(* Logix 5000 project; controller E2122_083_261121_V1 vendor 1 type 14 code 196 rev 32.11; software revision 32.00 *)

TASK MainTask (continuous, watchdog 500 ms) : MainProgram

MODULES
   Local : vendor 1 type 14 code 196 (5069 0, rev 32.11)
      HP : vendor 1 type 14 code 149 (Ethernet 192.168.4.220, rev 24.1, $01a7d3c3$ RPI 20 ms, $5cc36044$ RPI 20 ms, $f3259996$ RPI 20 ms, $494006c6$ RPI 20 ms, $5c112d50$ RPI 20 ms, $6e423aaa$ RPI 20 ms, $f0f89954$ RPI 20 ms, $571546d8$ RPI 20 ms, $782664ef$ RPI 20 ms, $0e272f01$ RPI 20 ms, $e1a11e23$ RPI 20 ms)
      RFID : vendor 322 type 12 code 102 (Ethernet 192.168.4.79, rev 1.1, StandardDataDriven RPI 10 ms)
      RFID_2 : vendor 322 type 12 code 102 (Ethernet 192.168.4.80, rev 1.1, StandardDataDriven RPI 10 ms)
       : 5069-IB16 (5069 1, rev 2.1, StandardDataDriven RPI 5 ms)
       : 5069-OB16 (5069 2, rev 2.1, StandardDataDriven RPI 5 ms)
END_MODULES

TYPE Createparams :
STRUCT
   Type : DINT;   // 1 for TCP , 2 for UDP
   Addr : SockAddr;
END_STRUCT
END_TYPE

TYPE OpenconnParams :
STRUCT
   Timeout : DINT;
   DestAddr : STRING;
END_STRUCT
END_TYPE

TYPE SOCK_Addr :
STRUCT
   Family : INT;   // Address Family Must be 2
   Port : INT;   // Port Number
   Addr : SINT[4];   // IP Address
END_STRUCT
END_TYPE

TYPE SOCK_CreateParams :
STRUCT
   Type : DINT;   // 1 - TCP 2- UPD
   Addr : SOCK_Addr;
END_STRUCT
END_TYPE

TYPE SOCK_DATA_CLIENT :
STRUCT
   Create_Source : SOCK_CreateParams;
   Instance : DINT;
   Connect_Source : SOCK_OpenConnParam;
   Read_Source : SOCK_ReadParams;
   Read_Response : SOCK_ReadResponse;
   Write_Source : SOCK_WriteParams;
   Write_SizeSent : DINT;
END_STRUCT
END_TYPE

TYPE SOCK_OpenConnParam :
STRUCT
   Timeout : DINT;
   DestAddr : STRING;
END_STRUCT
END_TYPE

TYPE SOCK_ReadParams :
STRUCT
   Timeout : DINT;
   BufLen : DINT;
END_STRUCT
END_TYPE

TYPE SOCK_ReadResponse :
STRUCT
   FromAddr : SOCK_Addr;
   Buffer : STRING_READBUFFER;
END_STRUCT
END_TYPE

TYPE SOCK_WriteParams :
STRUCT
   Timeout : DINT;
   ToAddr : SOCK_Addr;
   Buffer : STRING_WRITEBUFFER;
END_STRUCT
END_TYPE

TYPE SockAddr :
STRUCT
   Family : INT;   // 2 for IP4 family
   Port : INT;   // Port number
   Addr : DINT;   // Local IP = 0
END_STRUCT
END_TYPE

TYPE STR_480 :
STRUCT
   LEN : DINT;
   DATA : SINT[82];
END_STRUCT
END_TYPE

TYPE STRING_READBUFFER :
STRUCT
   LEN : DINT;
   DATA : SINT[484];
END_STRUCT
END_TYPE

TYPE STRING_WRITEBUFFER :
STRUCT
   LEN : DINT;
   DATA : SINT[462];
END_STRUCT
END_TYPE

TYPE WriteParams :
STRUCT
   Timeout : DINT;
   ToAddr : SockAddr;
   Buf : STR_480;
END_STRUCT
END_TYPE

ADD_ON_INSTRUCTION INACTIVE   (* revision 2.4 *)
VAR_INPUT
   iiChannelNo : INT; {required}   // channel-No. of DTE102
   ixConnOK : BOOL; {required}   // Ethernet/IP connection to DTE102 is OK
END_VAR
VAR_IN_OUT
   iarbDTE102 : SINT[80]; {required}   // input data from DTE102
   oarbDTE102 : SINT[80]; {required}   // output data to DTE102
END_VAR
VAR_INPUT
   ixAckDiag : BOOL; {required}   // acknowledge diagnostic data
END_VAR
VAR_OUTPUT
   oiDiagLength : INT; {access Read Only, required}   // number of diagnostic data
END_VAR
VAR_IN_OUT
   oardwDiagData : DINT[4]; {required}   // diagnostic data
END_VAR
VAR
   IChannelNo : INT; {access None}   // channel-No. set by ConnOK
   IActInputSize : INT; {access None}   // actual input data size of DTE102
   XConnOK : BOOL; {access None}   // connection OK
   IActOutputSize : INT; {access None}   // actual output data size of DTE102
   IDataOffset : INT; {access None}   // offset in DTE data
   XreIxAckDiag : BOOL; {access None}   // rising edge input acknowledge diagnostic data
   XprevIxAckDiag : BOOL; {access None}   // previous state of input acknowledge diagnostic data
   XInitDiag : BOOL; {access None}   // initialize output diagnostic data
   bStatusDTE : SINT; {access None}
   IRdIdx : INT; {access None}   // read index pointer
   XDrRdy : BOOL; {access None}   // read diagnostic data finished
   XDiag : BOOL; {access None}   // unread diagnostic data available
   IWrIdx : INT; {access None}   // write index pointer
END_VAR

ROUTINE Logic   (* structured text *)
   (*Disclaimer of Warranties
   ifm disclaims to the fullest extent authorized by law any and all warranties, whether express or implied, including,
   without limitation, any implied warranties of title, non-infringement, quiet enjoyment, integration, merchantability
   or fitness for a particular purpose.
   Without limitation of the foregoing, ifm expressly does not warrant that:
   (a) 	the software will meet your requirements or expectations;
   (b) 	the software or the software content will be free of bugs, errors, viruses or other defects;
   (c) 	any results, output, or data provided through or generated by the software will be accurate,
   	up-to-date, complete or reliable;
   (d) 	the software will be compatible with third party software;
   (e) 	any errors in the software will be corrected
   
   DEMO SOFTWARE AND TEMPLATES
   demo software and templates are provided “as is” and “as available”, without any warranty of any kind, either express or implied.
   The User acknowledges and agrees to use the software at User’s own risk. In no event shall ifm be held liable for any direct, indirect,
   incidental or consequential damages arising out of the use of or inability to use the software. User may use the software
   solely for demonstration purposes and to assess the software functionalities and capabilities.
   
   Software written specifically for Customer
   1. The software created and used is put together by ifm specially to the customer using modular
      software components made by ifm for numerous applications (Standard software modules) and adapted
      to the contractual service required (customer-specific application program).
   2. Upon complete payment of the purchase price for the customer-specific application program, ifm transfers
      the non-exclusive, locally and temporarily unrestricted usage right thereof to the customer, without the customer
      acquiring any rights of any kind to the standard software module on which the individual or customer-specific adaptation is based.
      Notwithstanding these provisions, ifm reserves the right to produce and offer customer specific software solutions of the same kind
      for other customers based on other terms of reference. In any case ifm retains a simple right of usage of the customer–specific
      solution for internal purposes.
   3. Upon acceptance of the program, User acknowledges and agrees to use the software at User’s own risk. User also acknowledges
      and agrees upon acceptance of the program that the software meets the requirements of the specifications agreed upon.
      ifm disclaims any and all warranties, in particular regarding fitness of the software for a particular purpose.
   *)
   
   case iiChannelNo of  (* check channel-No. *)
   1..4: (* channel-No. valid *)
     IChannelNo := iiChannelNo;  (* store channel-No. *)
   else  (* channel-No. invalid *)
     IChannelNo := 0;  (* mark as invalid channel-No. *)
   end_case;  (* check channel-No. *)
   
   XConnOK := (IChannelNo <> 0) and ixConnOK;  (* connection OK *)
   
   size(iarbDTE102,0,IActInputSize);  (* get input channel data size of DTE102 *)
   IActInputSize:= IActInputSize/4;
   size (oarbDTE102,0,IActOutputSize);  (* get output channel data size of DTE102 *)
   IActOutputSize:= IActOutputSize/4;
   
   
   XreIxAckDiag := ixAckDiag and not XprevIxAckDiag and not S:fs;  (* detect rising edge *)
   XprevIxAckDiag := ixAckDiag;  (* store state for detecting signal change *)
   
   if XConnOK and (IActInputSize = IActOutputSize) then  (* connection OK *)
   
     XInitDiag := XreIxAckDiag;  (* initialize output diagnostic data*)
   
     IDataOffset := IActInputSize * (IChannelNo - 1);  (* calculate offset for channel data *)
   
     (* check diagnostic data *)
     bStatusDTE := iarbDTE102[IDataOffset];  (* input byte 0 from DTE102 *)
     XDrRdy := bStatusDTE.6;  (* read diagnostic data finished *)
     XDiag  := bStatusDTE.7;  (* unread diagnostic data available *)
     oarbDTE102[IDataOffset].6 := XDiag and not XDrRdy;  (* read diagnostic data *)
     if XDiag and XDrRdy then  (* diagnostic data available *)
        cps (iarbDTE102[IDataOffset + 1],oiDiagLength,1); (* get number of diagnostic data *)
       IRdIdx := 2;  (* set index to data *)
       for IWrIdx := 0 to 3 do  (* loop all diagnostic data *)
         cps(iarbDTE102[IDataOffset + IRdIdx], oardwDiagData[IWrIdx],4);
         IRdIdx := IRdIdx + 4;  (* set read index to next diagnostic data *)
       end_for;  (* loop all diagnostic data *)
     end_if;  (* diagnostic data available *)
   
   else  (* connection failed *)
     XInitDiag := 0;  (* initialize output diagnostic data*)
   end_if;  (* connection OK *)
   
END_ROUTINE
END_ADD_ON_INSTRUCTION

ADD_ON_INSTRUCTION INPUT   (* revision 2.4 *)
VAR_INPUT
   iiChannelNo : INT; {required}   // channel-No. of DTE102
   ixConnOK : BOOL; {required}   // Ethernet/IP connection to DTE102 is OK
END_VAR
VAR_IN_OUT
   iarbDTE102 : SINT[80]; {required}   // input data from DTE102
   oarbDTE102 : SINT[80]; {required}   // output data to DTE102
END_VAR
VAR_INPUT
   ixAckDiag : BOOL; {required}   // acknowledge diagnostic data
END_VAR
VAR_OUTPUT
   oxCQi : BOOL; {access Read Only, required}   // status input C/Qi
   oxIQ : BOOL; {access Read Only, required}   // status input I/Q
   oxOverload : BOOL; {access Read Only, required}   // overload on L+
END_VAR
VAR_INPUT
   oiDiagLength : INT; {required}   // number of diagnostic data
END_VAR
VAR_IN_OUT
   oardwDiagData : DINT[4]; {required}   // iagnostic data
END_VAR
VAR
   IChannelNo : INT; {access None}   // channel-No. set by ConnOK
   IActInputSize : INT; {access None}   // actual input data size of DTE102
   XConnOK : BOOL; {access None}   // connection OK
   IActOutputSize : INT; {access None}   // actual output data size of DTE102
   IDataOffset : INT; {access None}   // offset in DTE data
   XreIxAckDiag : BOOL; {access None}   // rising edge input acknowledge diagnostic data
   XprevIxAckDiag : BOOL; {access None}   // previous state of input acknowledge diagnostic data
   XInitDiag : BOOL; {access None}   // initialize output diagnostic data
   bStatusDTE : SINT; {access None}
   IRdIdx : INT; {access None}   // read index pointer
   XDrRdy : BOOL; {access None}   // read diagnostic data finished
   XDiag : BOOL; {access None}   // unread diagnostic data available
   IWrIdx : INT; {access None}   // write index pointer
END_VAR

ROUTINE Logic   (* structured text *)
   (*Disclaimer of Warranties
   ifm disclaims to the fullest extent authorized by law any and all warranties, whether express or implied, including,
   without limitation, any implied warranties of title, non-infringement, quiet enjoyment, integration, merchantability
   or fitness for a particular purpose.
   Without limitation of the foregoing, ifm expressly does not warrant that:
   (a) 	the software will meet your requirements or expectations;
   (b) 	the software or the software content will be free of bugs, errors, viruses or other defects;
   (c) 	any results, output, or data provided through or generated by the software will be accurate,
   	up-to-date, complete or reliable;
   (d) 	the software will be compatible with third party software;
   (e) 	any errors in the software will be corrected
   
   DEMO SOFTWARE AND TEMPLATES
   demo software and templates are provided “as is” and “as available”, without any warranty of any kind, either express or implied.
   The User acknowledges and agrees to use the software at User’s own risk. In no event shall ifm be held liable for any direct, indirect,
   incidental or consequential damages arising out of the use of or inability to use the software. User may use the software
   solely for demonstration purposes and to assess the software functionalities and capabilities.
   
   Software written specifically for Customer
   1. The software created and used is put together by ifm specially to the customer using modular
      software components made by ifm for numerous applications (Standard software modules) and adapted
      to the contractual service required (customer-specific application program).
   2. Upon complete payment of the purchase price for the customer-specific application program, ifm transfers
      the non-exclusive, locally and temporarily unrestricted usage right thereof to the customer, without the customer
      acquiring any rights of any kind to the standard software module on which the individual or customer-specific adaptation is based.
      Notwithstanding these provisions, ifm reserves the right to produce and offer customer specific software solutions of the same kind
      for other customers based on other terms of reference. In any case ifm retains a simple right of usage of the customer–specific
      solution for internal purposes.
   3. Upon acceptance of the program, User acknowledges and agrees to use the software at User’s own risk. User also acknowledges
      and agrees upon acceptance of the program that the software meets the requirements of the specifications agreed upon.
      ifm disclaims any and all warranties, in particular regarding fitness of the software for a particular purpose.
   *)
   case iiChannelNo of  (* check channel-No. *)
   1..4: (* channel-No. valid *)
     IChannelNo := iiChannelNo;  (* store channel-No. *)
   else  (* channel-No. invalid *)
     IChannelNo := 0;  (* mark as invalid channel-No. *)
   end_case;  (* check channel-No. *)
   
   XConnOK := (IChannelNo <> 0) and ixConnOK;  (* connection OK *)
   
   size(iarbDTE102,0,IActInputSize);  (* get input channel data size of DTE102 *)
   IActInputSize:= IActInputSize/4;
   size (oarbDTE102,0,IActOutputSize);  (* get output channel data size of DTE102 *)
   IActOutputSize:= IActOutputSize/4;
   
   
   XreIxAckDiag := ixAckDiag and not XprevIxAckDiag and not s:fs;  (* detect rising edge *)
   XprevIxAckDiag := ixAckDiag;  (* store state for detecting signal change *)
   
   if XConnOK and (IActInputSize = IActOutputSize) then  (* connection OK *)
   
     XInitDiag := XreIxAckDiag;  (* initialize output diagnostic data*)
   
     IDataOffset := IActInputSize * (IChannelNo - 1);  (* calculate offset for channel data *)
   
     (* read status byte of DTE102 *)
     bStatusDTE := iarbDTE102[IDataOffset];  (* input byte 0 from DTE102 *)
     oxCQi := bStatusDTE.0;  (* input C/Qi *)
     oxIQ  := bStatusDTE.1;  (* input I/Q *)
     oxOverload  := bStatusDTE.3;  (* input overload *)
   
     (* check diagnostic data *)
     XDrRdy := bStatusDTE.6;  (* read diagnostic data finished *)
     XDiag  := bStatusDTE.7;  (* unread diagnostic data available *)
     oarbDTE102[IDataOffset].6 := XDiag and not XDrRdy;  (* read diagnostic data *)
     if XDiag and XDrRdy then  (* diagnostic data available *)
      cps (iarbDTE102[IDataOffset + 1],oiDiagLength,1); (* get number of diagnostic data *)
       IRdIdx := 2;  (* set index to data *)
       for IWrIdx := 0 to 3 do  (* loop all diagnostic data *)
         cps(iarbDTE102[IDataOffset + IRdIdx], oardwDiagData[IWrIdx],4);
         IRdIdx := IRdIdx + 4;  (* set read index to next diagnostic data *)
       end_for;  (* loop all diagnostic data *)
     end_if;  (* diagnostic data available *)
   
   else  (* connection failed *)
     XInitDiag := 1;  (* initialize output diagnostic data*)
     oxCQi := 0;  (* reset all outputs *)
     oxIQ  := 0;
     oxOverload  := 0;
   
   end_if;  (* connection OK *)
   
   if XInitDiag then  (* initialize output diagnostic data *)
     oiDiagLength := 0;
     oardwDiagData[0] := 0;
     oardwDiagData[1] := 0;
     oardwDiagData[2] := 0;
     oardwDiagData[3] := 0;
   end_if;  (* initialize output diagnostic data *)
   
END_ROUTINE
END_ADD_ON_INSTRUCTION

ADD_ON_INSTRUCTION OUTPUT   (* revision 2.4 *)
VAR_INPUT
   iiChannelNo : INT; {required}   // channel-No. of DTE102
   ixConnOK : BOOL; {required}   // Ethernet/IP connection to DTE102 is OK
END_VAR
VAR_IN_OUT
   iarbDTE102 : SINT[80]; {required}   // input data from DTE102
   oarbDTE102 : SINT[80]; {required}   // output data to DTE102
END_VAR
VAR_INPUT
   ixAckDiag : BOOL; {required}   // acknowledge diagnostic data
END_VAR
VAR_OUTPUT
   oxIQ : BOOL; {access Read Only, required}   // status input I/Q
   oxOverload : BOOL; {access Read Only, required}   // overload on L+
   oiDiagLength : INT; {access Read Only, required}   // number of diagnostic data
END_VAR
VAR_IN_OUT
   oardwDiagData : DINT[4]; {required}   // diagnostic data
END_VAR
VAR_INPUT
   ixCQo : BOOL; {required}   // output C/Qo
   ixHighCurrent : BOOL; {required}   // enable high current max. 1A (channel 3 and 4 onla)
END_VAR
VAR_OUTPUT
   oxCQi : BOOL; {access Read Only, required}
END_VAR
VAR
   IChannelNo : INT; {access None}   // channel-No. set by ConnOK
   IActInputSize : INT; {access None}   // actual input data size of DTE102
   XConnOK : BOOL; {access None}   // connection OK
   IActOutputSize : INT; {access None}   // actual output data size of DTE102
   IDataOffset : INT; {access None}   // offset in DTE data
   XreIxAckDiag : BOOL; {access None}   // rising edge input acknowledge diagnostic data
   XprevIxAckDiag : BOOL; {access None}   // previous state of input acknowledge diagnostic data
   XInitDiag : BOOL; {access None}   // initialize output diagnostic data
   bStatusDTE : SINT; {access None}   // status byte from DTE102
   bCmdDTE : SINT; {access None}   // command byte DTE102 (output byte 0
   IRdIdx : INT; {access None}   // read index pointer
   XDrRdy : BOOL; {access None}   // read diagnostic data finished
   XDiag : BOOL; {access None}   // unread diagnostic data available
   XDr : BOOL; {access None}   // read diagnostic data
   IWrIdx : INT; {access None}   // write index pointer
END_VAR

ROUTINE Logic   (* structured text *)
   (*Disclaimer of Warranties
   ifm disclaims to the fullest extent authorized by law any and all warranties, whether express or implied, including,
   without limitation, any implied warranties of title, non-infringement, quiet enjoyment, integration, merchantability
   or fitness for a particular purpose.
   Without limitation of the foregoing, ifm expressly does not warrant that:
   (a) 	the software will meet your requirements or expectations;
   (b) 	the software or the software content will be free of bugs, errors, viruses or other defects;
   (c) 	any results, output, or data provided through or generated by the software will be accurate,
   	up-to-date, complete or reliable;
   (d) 	the software will be compatible with third party software;
   (e) 	any errors in the software will be corrected
   
   DEMO SOFTWARE AND TEMPLATES
   demo software and templates are provided “as is” and “as available”, without any warranty of any kind, either express or implied.
   The User acknowledges and agrees to use the software at User’s own risk. In no event shall ifm be held liable for any direct, indirect,
   incidental or consequential damages arising out of the use of or inability to use the software. User may use the software
   solely for demonstration purposes and to assess the software functionalities and capabilities.
   
   Software written specifically for Customer
   1. The software created and used is put together by ifm specially to the customer using modular
      software components made by ifm for numerous applications (Standard software modules) and adapted
      to the contractual service required (customer-specific application program).
   2. Upon complete payment of the purchase price for the customer-specific application program, ifm transfers
      the non-exclusive, locally and temporarily unrestricted usage right thereof to the customer, without the customer
      acquiring any rights of any kind to the standard software module on which the individual or customer-specific adaptation is based.
      Notwithstanding these provisions, ifm reserves the right to produce and offer customer specific software solutions of the same kind
      for other customers based on other terms of reference. In any case ifm retains a simple right of usage of the customer–specific
      solution for internal purposes.
   3. Upon acceptance of the program, User acknowledges and agrees to use the software at User’s own risk. User also acknowledges
      and agrees upon acceptance of the program that the software meets the requirements of the specifications agreed upon.
      ifm disclaims any and all warranties, in particular regarding fitness of the software for a particular purpose.
   *)
   case iiChannelNo of  (* check channel-No. *)
   1..4: (* channel-No. valid *)
     IChannelNo := iiChannelNo;  (* store channel-No. *)
   else  (* channel-No. invalid *)
     IChannelNo := 0;  (* mark as invalid channel-No. *)
   end_case;  (* check channel-No. *)
   
   XConnOK := (IChannelNo <> 0) and ixConnOK;  (* connection OK *)
   size(iarbDTE102,0,IActInputSize);  (* get input channel data size of DTE102 *)
   IActInputSize:= IActInputSize/4;
   size (oarbDTE102,0,IActOutputSize);  (* get output channel data size of DTE102 *)
   IActOutputSize:= IActOutputSize/4;
   
   XreIxAckDiag := ixAckDiag and not XprevIxAckDiag and not S:fs;  (* detect rising edge *)
   XprevIxAckDiag := ixAckDiag;  (* store state for detecting signal change *)
   
   if XConnOK and (IActInputSize = IActOutputSize) then  (* connection OK *)
   
     XInitDiag := XreIxAckDiag;  (* initialize output diagnostic data*)
   
     IDataOffset := IActInputSize * (IChannelNo - 1);  (* calculate offset for channel data *)
   
     (* read status byte of DTE102 *)
     bStatusDTE := iarbDTE102[IDataOffset];  (* input byte 0 from DTE102 *)
     oxIQ  := bStatusDTE.1;  (* input I/Q *)
     oxCQi := bStatusDTE.0; (* input C/Qi *)
     oxOverload  := bStatusDTE.3;  (* input overload *)
   
     (* check diagnostic data *)
     XDrRdy := bStatusDTE.6;  (* read diagnostic data finished *)
     XDiag  := bStatusDTE.7;  (* unread diagnostic data available *)
     XDr := XDiag and not XDrRdy;  (* read diagnostic data *)
     if XDiag and XDrRdy then  (* diagnostic data available *)
        cps (iarbDTE102[IDataOffset + 1],oiDiagLength,1); (* get number of diagnostic data *)
       IRdIdx := 2;  (* set index to data *)
       for IWrIdx := 0 to 3 do  (* loop all diagnostic data *)
         cps(iarbDTE102[IDataOffset + IRdIdx], oardwDiagData[IWrIdx],4);
         IRdIdx := IRdIdx + 4;  (* set read index to next diagnostic data *)
       end_for;  (* loop all diagnostic data *)
     end_if;  (* diagnostic data available *)
   
      (* write command byte to DTE102 *)
     bCmdDTE := 0;  (* initialize command byte *)
     bCmdDTE.0 := ixCQo;
     bCmdDTE.2 := ixHighCurrent and (IChannelNo = 3 or IChannelNo = 4);  (* high current for channel 3 and 4 only *)
     bCmdDTE.6 := XDr;  (* request read diagnosis *)
     oarbDTE102[IDataOffset] := bCmdDTE;  (* set command byte to DTE102 *)
   
   else  (* connection failed *)
     XInitDiag := 1;  (* initialize output diagnostic data*)
   
     oxIQ := 0;  (* reset all outputs *)
     oxOverload  := 0;
   
   end_if;  (* connection OK *)
   
   if XInitDiag then  (* initialize output diagnostic data *)
     oiDiagLength := 0;
     oardwDiagData[0] := 0;
     oardwDiagData[1] := 0;
     oardwDiagData[2] := 0;
     oardwDiagData[3] := 0;
   end_if;  (* initialize output diagnostic data *)
   
END_ROUTINE
END_ADD_ON_INSTRUCTION

ADD_ON_INSTRUCTION RWH_RW   (* revision 2.4, vendor ifm syntron *)
// Read/Write AddOn for DTE102
// Revision note:
// resolved the speed issue causedby usage of for loops.
VAR_INPUT
   ixConnOK : BOOL; {required}   // Ethernet/IP connection to DTE102 is OK
   iiChannelNo : INT; {required}   // channel-No. set by ConnOK
   ixRead : BOOL; {required}   // read data from tag
   ixWrite : BOOL; {required}   // write data to tag
END_VAR
VAR_OUTPUT
   oxBusy : BOOL; {access Read Only, required}   // command in progress
END_VAR
VAR_IN_OUT
   oarbDTE102 : SINT[80]; {required}   // output data to DTE102
   iarbDTE102 : SINT[80]; {required}   // input data from DTE102
END_VAR
VAR_INPUT
   ixUserMem : BOOL; {required}   // access to USER memory on tag
   ixAntOff : BOOL; {required}   // deactivate antenna
   iiRdWrLength : INT; {required}   // data length (in BYTEs) to read/write USER memory on tag
   iiRdWrStartAddr : INT; {required}   // start address to read/write USER memory on tag
END_VAR
VAR_IN_OUT
   iarbSendBuf : SINT[32]; {required}   // send buffer for data to write to USER memory on tag
   oarbRcvBuf : SINT[32]; {required}   // receive buffer for data from tag
   oardwDiagData : DINT[4]; {required}   // diagnostic data
END_VAR
VAR_OUTPUT
   oxError : BOOL; {access Read Only, required}   // error occurred
   oxDone : BOOL; {access Read Only, required}   // command completed without error
   oiRcvdLength : INT; {access Read Only, required}   // data length (in BYTEs) read from the tag
   owStatus : DINT; {access Read Only, required}   // status
   oxTagPresent : BOOL; {access Read Only, required}   // tag present
   oiDiagLength : INT; {access Read Only, required}   // number of diagnostic data
END_VAR
VAR
   XConnOK : BOOL; {access None}   // rising edge of connection OK
   XStartupPLC : BOOL; {access None}   // plc first task run
   XreConnOK : BOOL; {access None}   // rising edge of connection OK
   XprevConnOK : BOOL; {access None}   // previous state of connection OK
   IChannelNo : INT; {access None}   // channel-No. of DTE102
   IInputSize : INT; {access None}   // input data size of DTE102
   IActDteInputSize : INT; {access None}   // actual input data size of DTE102
   IOutputSize : INT; {access None}   // output data size of DTE102
   IActDteOutputSize : INT; {access None}   // actual output data size of DTE102
   ISendBufSize : INT; {access None}   // send buffer size (in BYTE)
   IActSendBufSize : INT; {access None}   // actual send buffer size (in BYTE)
   IRcvBufSize : INT; {access None}   // receive buffer size (in BYTE)
   IActRcvBufSize : INT; {access None}   // actual receive buffer size (in BYTE)
   IState : INT; {access None}   // sequence pointer
   IDataOffset : INT; {access None}   // offset for channel data of DTE102
   bStatusDTE : SINT; {access None}   // status byte from DTE102 (input byte 0)
   bCmdDTE : SINT; {access None}   // command byte DTE102 (output byte 0)
   IRdWrStartAddr : INT; {access None}   // start address to read or write
   XErrorSettings : BOOL; {access None}   // error in settings
   WErrorCode : DINT; {access None}   // error code
   XreIxRead : BOOL; {access None}   // rising edge input read
   XprevIxRead : BOOL; {access None}   // previous state of input read
   XreIxWrite : BOOL; {access None}   // rising edge input write
   XprevIxWrite : BOOL; {access None}   // previous state of input write
   XUserAction : BOOL; {access None}   // user action started
   XError : BOOL; {access None}   // error occurred
   IParamSize : INT; {access None}   // max. parameter length in I/O-data of DTE102
   ILeftCycles : INT; {access None}   // left read or write cycles to do
   XTp : BOOL; {access None}   // tag present
   XAi : BOOL; {access None}   // antenna inactive
   XWrRdy : BOOL; {access None}   // writing data finished
   XRdRdy : BOOL; {access None}   // reading data finished
   XUd : BOOL; {access None}   // user memory register is open
   XDrRdy : BOOL; {access None}   // read diagnostic data finished
   XDiag : BOOL; {access None}   // unread diagnostic data available
   XAo : BOOL; {access None}   // switch off antenna
   XWr : BOOL; {access None}   // write data
   XRd : BOOL; {access None}   // read data
   XUr : BOOL; {access None}   // open user memory register
   XDr : BOOL; {access None}   // read diagnostic data
   TonTimeout : FBD_TIMER; {access None}   // command time out
   XWrExec : BOOL; {access None}   // writing command executed
   TonDlyInit : FBD_TIMER; {access None}   // delay initialisation sequence
   IDataLength : INT; {access None}   // length to read or write (in BYTE)
   IRdIdx : INT; {access None}   // read index pointer
   IWrIdx : INT; {access None}   // write index pointer
   IRdLengthTotal : INT; {access None}   // read length total
   XKeepOutput : BOOL; {access None}   // keep outputs active
   ITempHighByte : INT; {access None}   // temporary flag to sore high byte
   IActChInputSize : INT; {access None}
   IActChOutputSize : INT; {access None}
   XFinished : BOOL; {access None}
   XDteAction : BOOL; {access None}
END_VAR

ROUTINE Logic   (* structured text *)
   XStartupPLC:= s:fs; // plc first task run
   
   //************************************
   //**** get array sizes ****
   
   size(iarbDTE102,0,IActDteInputSize);  // get input size of DTE102
   IActChInputSize:= IActDteInputSize/4; // calculate input channel size
   size (oarbDTE102,0,IActDteOutputSize);  // get output size of DTE102
   IActChOutputSize:= IActDteOutputSize/4; // calculate output channel size
   size(iarbSendBuf,0,IActSendBufSize);  // get send buffer size
   size(oarbRcvBuf,0,IActRcvBufSize);  // get receive buffer size
   
   //******************************
   //** check settings parameter **
   
   XConnOK := ixConnOK and not XStartupPLC;  // not at startup plc
   XreConnOK := XConnOK and not XprevConnOK;  // detecting rising edge
   XprevConnOK := XConnOK;  // store state for detecting signal change
   
   if XreConnOK then  // freeze settings on rising edge of connection OK
     case iiChannelNo of  // freeze channel-No.
     1..4: // channel-No. valid
       IChannelNo := iiChannelNo;  // store channel-No.
     else  // channel-No. invalid
       IChannelNo := 0;  // mark as invalid channel-No.
     end_case;  // freeze channel-No.
     IInputSize := IActChInputSize;  // freeze actual array sizes
     IOutputSize := IActChOutputSize;
     ISendBufSize := IActSendBufSize;
     IRcvBufSize := IActRcvBufSize;
   end_if;  // freeze settings on rising edge of connection OK
   
   if XConnOK then  // watch settings parameters
     if (IChannelNo = 0) or (IChannelNo <> iiChannelNo) then  // check parameter Channel
       XErrorSettings := 1;  // set error in settings parameter
   // error code 8101
       WErrorCode := 16#8101;  // set error code
     elsif (IActChInputSize * 4 <> IActDteInputSize) or (IInputSize <> IActChInputSize) then  // check parameter input from DTE102
       XErrorSettings := 1;  // set error in settings parameter
   // error code 8102
       WErrorCode := 16#8102;  // set error code
     elsif (IActChOutputSize * 4 <> IActDteOutputSize) or (IOutputSize <> IActChOutputSize) then  // check parameter output to DTE102
       XErrorSettings := 1;  // set error in settings parameter
   // error code 8103
       WErrorCode := 16#8103;  // set error code
     elsif IInputSize <> IOutputSize then  // check parameter input and output size to DTE102
       XErrorSettings := 1;  // set error in settings parameter
   // error code 8104
       WErrorCode := 16#8104;  // set error code
     elsif (ISendBufSize <> IActSendBufSize) then  // check parameter send buffer
       XErrorSettings := 1;  // set error in settings parameter
   // error code 8105
       WErrorCode := 16#8105;  // set error code
     elsif (IRcvBufSize <> IActRcvBufSize) then  // ckeck parameter receive buffer
       XErrorSettings := 1;  // set error in settings parameter
   // error code 8106
       WErrorCode := 16#8106;  // set error code
     else  // no connection
       XErrorSettings := 0;  // reset error in settings parameter
     end_if;  // error list
   end_if;  // watch settings parameters
   
   
   //*************************
   //** check input signals **
   
   XreIxRead := ixRead and not XprevIxRead and not XStartupPLC;  // detect rising edge
   XprevIxRead := ixRead;  // store state for detecting signal change
   
   XreIxWrite := ixWrite and not XprevIxWrite and not XStartupPLC;  // detect rising edge
   XprevIxWrite := ixWrite;  // store state for detecting signal change
   
   if XreIxRead or XreIxWrite then  // detect user action
     XUserAction := 1;  // set user action started
     if oxBusy and not XError then  // command active already
       XError := 1;  // set error occurred
   // error code 8301
       WErrorCode := 16#8301;  // set error code
     end_if;  // Command active already
   end_if;  // detect user action
   
   if not XConnOK and XUserAction and not XStartupPLC then  // connection lost while user action in progress
     if not XError then  // no error occurred yet
       XError := 1;  // set error occurred
   // error code 8201
       WErrorCode := 16#8201;  // set error code
     end_if;  // no error occurred yet
   end_if;  // connection lost while user action in progress
   
   if not XConnOK or XErrorSettings then  // connection to DTE fail
   
     XUserAction := 0;  // reset user action started
     IState := 16#1000;  // initialize main sequence
   
   else  // connection to DTE102 OK
   
     IDataOffset := IInputSize * (IChannelNo - 1);  // calculate offset for channel data
   
   // read status byte of DTE102
     bStatusDTE := iarbDTE102[IDataOffset];  // input byte 0 from DTE102
     XTp    := bStatusDTE.0;  // tag present
     XAi    := bStatusDTE.1;  // antenna inactive
     XWrRdy := bStatusDTE.2;  // write data to USER memory finished
     XRdRdy := bStatusDTE.3;  // read UID or USER memory data finished
     XUd    := bStatusDTE.4;  // USER memory mode active
     XDrRdy := bStatusDTE.6;  // read diagnostic data finished
     XDiag  := bStatusDTE.7;  // unread diagnostic data available
   
   // read command byte from DTE102
     bCmdDTE := oarbDTE102[IDataOffset];  // output byte 0 to DTE102
     XAo := bCmdDTE.1;  // switch off antenna
     XWr := bCmdDTE.2;  // write data
     XRd := bCmdDTE.3;  // read data
     XUr := bCmdDTE.4;  // activate USER memory mode
     XDr := bCmdDTE.6;  // read diagnostic data
   
   
   //**************
   //** time out **
   
   XDteAction:= (XUr xor XUd)
     	  		 or  (XWr xor XWrRdy)
   	  		 or  (XRd xor XRdRdy)
   	 		or  (XDr xor XDrRdy);
   
   
   TonTimeout.Reset:= not( XDteAction and XUserAction);
   
   
     TonTimeout.PRE := 700;  // set timeout time
     TonTimeout.TimerEnable :=  XDteAction and XUserAction;
     TONR(TonTimeout);
   
     if TonTimeout.DN then  // timeout occurred
       TonDlyInit.Reset:= 1;
   	if not XError then  // no error occurred yet
         XError := 1;  // set error occurred
   // error code 8202
         WErrorCode := 16#8202;  // set error code
       end_if;  // no error occurred yet
       IState := 16#1000;
     end_if;  // timeout occurred
   
   
   //*******************
   //** main sequence **
   
   	TonDlyInit.Reset :=  not(    ((XUr and XUd)or(not XUr and not XUd))
   		   				     and ((XAo and XAi) or (not XAo and not XAi)));
   
   
   
     case IState of
   
     16#1000: // wait for connection OK
   	    TonDlyInit.PRE:= 200;//preset timer to 200 ms
   		TonDlyInit.TimerEnable:=     ((XUr and XUd)or(not XUr and not XUd))
   		  						 and ((XAo and XAi) or (not XAo and not XAi)); // Enable Timer
   	    TONR(TonDlyInit);
   
   	  	XUr := XUd;  // set outputs to actual status of DTE
           XAo := 0;  // activate antenna
   		XWr := 0;  // write data
     		XRd := 0;  // read data
     		XDr := 0;  // read diagnostic data
   
   		if TonDlyInit.DN then
   	      IState := 16#2000;  // switch antenna off
   		end_if;
   
     16#2000: // check input signals from DTE102
    		 COP(oarbDTE102[IDataOffset + 1], oarbDTE102[IDataOffset], IWrIdx);
   		 IWrIdx := IOutputSize;
   		 if XDiag then  // diagnostic data available
   	       IState := 16#2402;  // read diagnostic data
   	     elsif XRdRdy then  // cancel active read function by send new
   	       XUr := 1;  // activate USER memory mode
      	       IState := 16#2101;  // read data
   	     elsif XWrRdy then  // cancel active write function by send new
   	       XUr := 1;  // activate USER memory mode
   	       IState := 16#2201;  // switch off antenna for not writing on tag
   		 else  // no active function
   	       IState := 16#3000;  // check antenna on/off
   	     end_if;  // diagnostic data available
   
   
   //***********************************
   //** initialize read data function **
   
     16#2101: // wait for USER memory mode active
              if XUd then  // USER memory mode active
                IState := 16#2102;  // set read command
              end_if;  // USER memory mode active
   
     16#2102: // wait diagnostic event
              if XDiag then  // diagnosic data appeared
   	     IState := 16#2103;  // reaet read command
              end_if;  // diagnosic data appeared
   
     16#2103: // complete read function
              if not XRdRdy then  // read data finished
   		     IState := 16#2402;  // set read diag command
   		   end_if;  // read data finished
   
   
   //*******************************************
   //** initialize write data function **
   
     16#2201: // wait for USER memory mode active
              if XUd then  // USER memory mode active
                IState := 16#2202;  // set write command
              end_if;  // USER memory mode active
   
     16#2202: // wait diagnostic event
              if XDiag then  // diagnosic data appeared
   	         IState := 16#2203;  // reset write command
              end_if;  // diagnosic data appeared
   
     16#2203: // complete write function
              if not XWrRdy then  // write data finished
   	         IState := 16#2402;  // set read diag command
   	       end_if;  // write data finished
   
   
   //********************************
   //** initialize diagnostic data **
   
     16#2402: // read diagnostic data
              if XDrRdy then  // read diagnostic data finished
                IState := 16#2403;  // reset read diag command
   	       end_if;  // read diagnostic data finished
   
     16#2403: // complete read diagnostic data
              if not XDrRdy then  // read diagnostic data finished
                if XDiag then  // still diagnostic data available
   	           IState := 16#2402;  // set read diag command
   	         else  // no diagnostic data available
   	           IState := 16#2000;  // check signals
   	         end_if;  // still diagnostic data available
   	       end_if;  // read diagnostic data finished
   
   
   //*****************
   //** antenna off **
   
     16#3000: // antenna off
   		if (XUr and XUd) or (not XUr and not XUd) then // mode steady
   	     XAo := ixAntOff;  // antenna off/on
              end_if;// mode steady
   
   	   if (XAo and XAi) or (not XAo and not XAi) then // antenna steady
   	     XUr := ixUserMem;  // (de)activate USER memory mode
   	   end_if; // antenna steady
   	   if XDiag then  // diagnostic data available
   	     IState := 16#7401;  // read diagnostic data
   	   elsif not XAo and not XAi then  // antenna not inactive
   	     IState := 16#7000;  // start normal operation mode
   	   end_if;  // diagnostic data available
   
   
   
   
   //***************************
   //** normal operation mode **
   
     16#7000: // wait for command
   
   	   if (XUr and XUd) or (not XUr and not XUd) then // mode steady
   	     XAo := ixAntOff;  // antenna off/on
              end_if; // mode steady
   
   	   if (XAo and XAi) or (not XAo and not XAi) then // antenna mode steady
   	     XUr := ixUserMem;  // (de)activate USER memory mode
   	   end_if; // antenna mode steady
   
   	   XWrExec := (XreIxWrite or XWrExec) and not XreIxRead; // execute writing command
   
   // diagnostic data available
            if XDiag then
   	     IState := 16#7401;  // read diagnostic data
   
   	   // if switch antenna off
            elsif XAo or XAi then
   	     if (XreIxRead or XreIxWrite) and not XError then  // no error occurred yet
   	       XError := 1;  // set error occurred
   // error code 8302
                WErrorCode := 16#8302;  // set error code
   	       end_if;  // no error occurred yet
    	       IState := 16#3000;  // wait for antenna on
   
              // read and write command at the same time
   	     elsif XreIxRead and XreIxWrite then
              if not XError then  // no error occurred yet
   	         XError := 1;  // set error occurred
   
   // error code 8303
   	       WErrorCode := 16#8303;  // set error code
   	       end_if;  // no error occurred yet
   
   
   // read or write command while no tag in field
   	   elsif (XreIxRead or XreIxWrite) and not XTp then
                if not XError then  // no error occurred yet
   	       XError := 1;  // set error occurred
   
   // error code 8304
   	       WErrorCode := 16#8304;  // set error code
   	     end_if;  // no error occurred yet
   
   // start read USER memory
   	   elsif XreIxRead and ixUserMem then
   	     if (iiRdWrLength <= 0) or (iiRdWrLength > IRcvBufSize) then  // read length parameter invalid
                  if not XError then  // no error occurred yet
   	         XError := 1;  // set error occurred
   // error code 8305
   	         WErrorCode := 16#8305;  // set error code
   	       end_if;  // no error occurred yet
                else  // read length parameter valid
   	        IRdWrStartAddr := iiRdWrStartAddr;  // save start address parameter
   	        IParamSize := IInputSize - 4;  // calculate max. data length in input data
   	        ILeftCycles := iiRdWrLength / IParamSize;  // left cycles with max. data length to do
   	        IDataLength := iiRdWrLength mod IParamSize;  // length to read in first cycle
               if IDataLength = 0 then  // only full parameter data to use
   	          IDataLength := IParamSize;  // set length to read in first cycle to max. data length
   		      ILeftCycles := ILeftCycles - 1;  // 1 less left cycle with max. data length to do
   	        end_if;  // only full parameter data to use
   	        cps(IDataLength,oarbDTE102[IDataOffset + 1],1); // set data length in command
   	        oarbDTE102[IDataOffset + 2]:= 0;
   	        ITempHighByte:= IRdWrStartAddr/256;
   		    cps (ITempHighByte,oarbDTE102[IDataOffset + 2],1);
   		    cps (IRdWrStartAddr, oarbDTE102[IDataOffset + 3],1);// low-byte of start address on tag
   	        if not XUd then  // USER memory mode inactive
   	          IState := 16#7101;  // wait USER memory mode
   	        else  // USER memory mode active
   	          IState := 16#7102;  // read data
               end_if;  // USER memory mode inactive
   	     end_if;  // read length parameter invalid
   
   	   // start write USER memory
   	     elsif XreIxWrite and ixUserMem then
   	       if (iiRdWrLength <= 0) or (iiRdWrLength > ISendBufSize) then  // write length parameter invalid
                if not XError then  // no error occurred yet
   	           XError := 1;  // set error occurred
   // error code 8306
   	           WErrorCode := 16#8306;  // set error code
   	         end_if;  // invalid write length parameter
   	       else  // write length parameter valid
   	         IRdWrStartAddr := iiRdWrStartAddr;  // save start address parameter
   	         IParamSize := IOutputSize - 4;  // calculate max. data length in output data
   	         ILeftCycles := iiRdWrLength / IParamSize;  // left cycles with max. data length to do
   	         IDataLength := iiRdWrLength mod IParamSize;  // length to write in first cycle
                if IDataLength = 0 then  // only full parameter data to use
   	           IDataLength := IParamSize;  // set length to write in first cycle to max. data length
   		       ILeftCycles := ILeftCycles - 1;  // 1 less left cycle with max. data length to do
   	         end_if;  // only full parameter data to use
   	         cps (IDataLength, oarbDTE102[IDataOffset + 1],1); // set data length in command
   	         ITempHighByte:= IRdWrStartAddr/256;
   		     cps (ITempHighByte,oarbDTE102[IDataOffset + 2],1);
   		     cps (IRdWrStartAddr, oarbDTE102[IDataOffset + 3],1);
   	         IRdIdx := 0;  // set read index to begin of send buffer
   	         for IWrIdx := 4 to IDataLength + 3 do  // loop all data to write in this write cycle
   	           oarbDTE102[IDataOffset + IWrIdx] := iarbSendBuf[IRdIdx];  // transfer data from send Buffer
   	           IRdIdx:=(IRdIdx +1 );  // update read index in send buffer
   	         end_for;  // loop all data to write in this write cycle
   	         if not XUd then  // USER memory mode inactive
   	           IState := 16#7201;  // wait USER memory mode
   	         else  // USER memory mode active
   	           IState := 16#7202;  // write data
                end_if;  // USER memory mode inactive
   	     end_if;  // USER memory mode inactive
   
   	   // start read UID
            elsif XreIxRead and not ixUserMem then
   	     // initialize parameter data in output to DTE102
   		 	 oarbDTE102[IDataOffset + 1] := 0;
   			 IWrIdx := IOutputSize - 1;
   			 COP(oarbDTE102[IDataOffset + 1], oarbDTE102[IDataOffset + 2], IWrIdx);
   			 IWrIdx := IOutputSize;
   	       if XUd then  // USER memory mode active
   	         IState := 16#7301;  // deactivate USER memory mode
   	       else  // USER memory mode not active
   	         IState := 16#7302;  // read data
              end_if; // USER memory mode active
   
   
   	   // invalid signal combination
   	     elsif XreIxWrite and not ixUserMem then  // write UID not possible
              if not XError then  // no error occurred yet
   	         XError := 1;  // set error occurred
   // error code 8307
   	         WErrorCode := 16#8307;  // set error code
   	       end_if;  // no error occurred yet
   
   
            end_if;  // end of command list
   
   
   //************************************
   //**** read USER memory ****
   
     16#7101: // wait for USER memory mode
              if XUd then  // USER memory mode active
                IState := 16#7102;  // read USER data
              end_if;  // USER memory mode active
   
     16#7102: // read USER data
               if XRdRdy then  // read data available
                if not XDiag and not XError then  // transfer data only if no error occurred yet
   			   COP(iarbDTE102[IDataOffset + 2], oarbRcvBuf[IWrIdx], IDataLength);
   			   IRdIdx := IDataLength + 1;
   			   IWrIdx := IWrIdx + IDataLength;
         	       IRdLengthTotal := IRdLengthTotal + IDataLength;  // store total received length
   	         end_if;  // transfer data only if no error occurred yet
                IState := 16#7103;  // complete read cycle
              end_if;  // read data available
   
   
     16#7103: // complete read cycle
             if not XRdRdy then  // reading data finished
   	        if XDiag then  // DTE error occurred
   	          IState := 16#7402;  // read diagnostic data
   	        else  // no DTE error occurred
   	          if (ILeftCycles > 0) and not XError then  // more data to read
   	            ILeftCycles := ILeftCycles - 1;  // decrease number of left cycles to do
   	            IRdWrStartAddr := IRdWrStartAddr + IDataLength;  // calculate next start address on tag
   	            IDataLength := IParamSize;  // set data length to maximum
   	            cps (IDataLength, oarbDTE102[IDataOffset + 1],1); // read max. length in following cycles
     			    ITempHighByte:= IRdWrStartAddr/256;
   		        cps (ITempHighByte,oarbDTE102[IDataOffset + 2],1);
   		        cps (IRdWrStartAddr, oarbDTE102[IDataOffset + 3],1);
   	            IState := 16#7102;  // read USER data
   	          else  // no more data to read
   	            IState := 16#7000;  // read USER data finished
   	          end_if;  // more data to read
   	        end_if;  // DTE error occurred
   	      end_if;  // reading data finished
   
   
   //************************************
   //**** write USER memory ****
   
     16#7201: // wait for USER memory mode
              if XUd then  // USER memory mode active
                IState := 16#7202;  // write USER data
              end_if;  // USER memory mode active
   
     16#7202: // write USER data
              if XWrRdy then  // write data finished
   	     IState := 16#7203;  // write USER data finished
              end_if;
   
     16#7203: // complete write cycle
            if not XWrRdy then  // writing data finished
   	       if XDiag then  // DTE error occurred
   	         IState := 16#7402;  // read diagnostic data
   	       else  // no DTE error occurred
   	         if (ILeftCycles > 0) and not XError then  // more data to write
   	           ILeftCycles := ILeftCycles - 1;  // decrease number of left cycles to do
   	           IRdWrStartAddr := IRdWrStartAddr + IDataLength;  // calculate next start address on tag
   	           IDataLength := IParamSize;  // set data length to maximum
   	           cps (IDataLength, oarbDTE102[IDataOffset + 1],1); // set data length in command
   			   ITempHighByte:= IRdWrStartAddr/256;
   		       cps (ITempHighByte,oarbDTE102[IDataOffset + 2],1);
   		       cps (IRdWrStartAddr, oarbDTE102[IDataOffset + 3],1);
   	           for IWrIdx := 4 to IDataLength + 3 do  // loop all data to write in this write cycle
   	             oarbDTE102[IDataOffset + IWrIdx] := iarbSendBuf[IRdIdx];  // transfer data from send Buffer
   	             IRdIdx:= IRdIdx +1;  // update read index in send buffer
   	           end_for;
   	           IState := 16#7202;  // write USER data
   	         else  // no more data to write
   	           IState := 16#7000;  // write USER data finished
   	         end_if;  // more data to write
   	       end_if;  // DTE error occurred
   	     end_if;  // writing data finished
   
   
   //*******************
   //** read UID data **
   
     16#7301: // wait for USER memory mode inactive
              if not XUd then  // USER memory mode inactive
                IState := 16#7302;  // read UID data
              end_if;
   
     16#7302: // read UID data
              if XRdRdy then  // read UID data finished
                if not XDiag and not XError then  // transfer data only if no error occurred yet
                  IDataLength := ( iarbDTE102[IDataOffset + 1]);  // get length of UID data
                  if IDataLength > IRcvBufSize then  // receive buffer too small
                    if not XError then  // no error occurred yet
   	           XError := 1;  // set error occurred
   // error code 8401
   	           WErrorCode := 16#8401;  // set error code
   	         end_if;  // no error occurred yet
                  else  // enough receive buffer
                    COP(iarbDTE102[IDataOffset + 2], oarbRcvBuf[0], IDataLength);// transfer UID into receive buffer
                    IWrIdx:= IDataLength -1 ;
   				 IRdLengthTotal := IDataLength;  // store received length
                  end_if;  // receive buffer too small
   	         end_if;  // transfer data only if no error occurred yet
        	     IState := 16#7303;  // complete read UID
              end_if;  // read UID data finished
   
     16#7303: // complete read UID
             if not XRdRdy then  // read finished
   	        if XDiag then  // DTE error occurred
   	          IState := 16#7402;  // read diagnostic data
   	        else  // no DTE error occurred
                  IState := 16#7000;  // function finished
   	        end_if;  // DTE error occurred
   	      end_if;  // read finished
   
   
   //**************************
   //** read diagnostic data **
   
     16#7401: // wait for USER memory mode (de)activated
           if (not XUd and not XUr)or (XUd and XUr) then // mode steady
   	     IState := 16#7402;  // read diagnistic data
   		end_if;  // mode steady
   
     16#7402: // read diagnostic data
           if XDrRdy or (not XDiag and XAi)  then  // read diagnostic data finished
           	if XUserAction and not XError then  // no error occurred yet
   	       		XError := 1;  // set error occurred
   // error code 8000
   				WErrorCode := 16#8000;  // set error code
   	    	end_if;  // no error occurred yet
   	     oiDiagLength := ( iarbDTE102[IDataOffset + 1]);  // get number of diagnostic data
   	     IRdIdx := 2;  // set index to data
   	     for IWrIdx := 0 to 3 do  // loop all diagnostic data
   	      cps(iarbDTE102[IDataOffset + IRdIdx], oardwDiagData[IWrIdx],4);
             IRdIdx := IRdIdx + 4;  // set read index to next diagnostic data
   	     end_for;  // loop all diagnostic data
   	     IState := 16#7403;  // complete read diagnostic data
   	   end_if;
   
     16#7403: // complete read diagnostic data
              if not XDrRdy then  // read diagnostics completed
   	     IState := 16#7000;  // function finished
              end_if;  // read diagnostics completed
   
    	  else  // case
      	 IState := 16#1000;  // initialize state
     end_case;
   
   
   //*********************************
   //** redirect state by antenna off
   
   XFinished := IState = 16#7000;  // function finished
   if XFinished and ixAntOff then  // redirect state
     XAo := 1;  // switch off antenna
     IState := 16#3000;  // antenna off
   end_if;  // redirect state
   
   
   //*********************
   //** set DTE outputs **
   
     // write command byte to DTE102
       bCmdDTE := 0;  // initialize command byte
   	bCmdDTE.1 := XAo;  // switch antenna off
       bCmdDTE.2 := (IState = 16#2202) or (IState = 16#7202);  // request write data
       bCmdDTE.3 := (IState = 16#2102) or (IState = 16#7102) or (IState = 16#7302);  // request read UID or user data
       bCmdDTE.4 := XUr;  // activate USER memory mode
       bCmdDTE.6 := (IState = 16#2402) or (IState = 16#7402);  // request read diagnosis
       oarbDTE102[IDataOffset] := bCmdDTE;  // set command byte to DTE102
   
   end_if;  // connection to DTE OK
   
   
   //*********************
   //** set DFB outputs **
   
   XKeepOutput := (ixRead and not XWrExec or ixWrite and XWrExec)  // input still active
   	    and not XreIxRead and not XreIxWrite and not XStartupPLC;  // until new command
   
   oxBusy := IState <> 16#7000;  // not ready for new command
   
   oxError := XError and (IState <= 16#7000)or XErrorSettings  // error occurred
           or oxError and XKeepOutput;  // keep output signal as long input active
   
   
   
   
   oxDone := (XUserAction and XFinished and not oxError)  // set function finisched without error
          or oxDone and XKeepOutput;  // keep output signal as long input is active
   
   
   
   
   
   if oxDone then  // function successfull finished
     owStatus := 0;  // output Status = 0x0000
     oiRcvdLength := IRdLengthTotal;  // show received length total
   
   elsif oxError then  // error occurred
     XError := 0;  // reset signal error occurred
     owStatus := WErrorCode;  // show error code
   else  // show status
     owStatus := IState;  // show state of sequence
   end_if;
   
   oxTagPresent := XTp and not XAi and XConnOK and not XErrorSettings;  // show tag present
   
   if (IState <= 16#7000) or oxError then  // no function in progress
     XUserAction := 0;  // reset user action started
   end_if;  // function in progress
   
   //*****************************************************
   // initialize receive buffer or show cyclic UID data **
   
   if oxError or XreIxRead or XreIxWrite or not XConnOK or (XAi and not oxDone) then  // initialize receive buffer
     for IWrIdx := 0 to IRcvBufSize - 1 do  // loop complete receive buffer
       oarbRcvBuf[IWrIdx] := 0;  // initialize receive buffer entry
     end_for;  // loop complete receive buffer
     IWrIdx := 0;  // set write index to begin
     IRdLengthTotal := 0;  // initialize received data length
     oiRcvdLength := 0;  // update output received length
   elsif not (oxBusy or oxDone) then  // check cyclic UID data
     IDataLength := (iarbDTE102[IDataOffset + 1]);  // get length in input data
     if IDataLength > IRcvBufSize then  // receive buffer too small
       oxError := 1;  // show error
   // error code 8401
       owStatus := 16#8401;  // show error code
     else  // enough receive buffer
       IParamSize := IInputSize - 4;  // calculate max. data length in input data
        for IWrIdx := 0 to IRcvBufSize - 1 do  // loop complete receive buffer
       	if IWrIdx < IParamSize then
   			oarbRcvBuf[IWrIdx] := iarbDTE102[IDataOffset + IWrIdx +2];  // Transfer UID into receive buffer
   		else
   			oarbRcvBuf[IWrIdx] := 0; // initialize receive buffer data
   		end_if;
   	 end_for;  // loop complete receive buffer
   	(*COP(iarbDTE102[IDataOffset +2], oarbRcvBuf[0], IParamSize);*)
   	IWrIdx := IRcvBufSize -1;
   	oiRcvdLength := IDataLength; // show UID length
     end_if;  // receive buffer too small
   end_if;  // initialize receive buffer or check cyclic UID data
   
   
   //********************************
   //** initialize diagnostic data **
   
   if XreIxRead or XreIxWrite or not XConnOK then  // initialize diagnostic data
     oiDiagLength := 0;  // initialize diagnostic data
     oardwDiagData[0] := 0;
     oardwDiagData[1] := 0;
     oardwDiagData[2] := 0;
     oardwDiagData[3] := 0;
   end_if;  // initialize diagnostic data
   
   
   
END_ROUTINE
END_ADD_ON_INSTRUCTION

VAR_GLOBAL   (* controller tags *)
   ACCEPT_PB_OP30 : ALIAS FOR Local:1:I.Pt00.Data;
   ACT_PR_STN4 : REAL;
   AntOffCh1 : BOOL;
   AntOffCh1_STN1 : BOOL;
   AntOffCh2 : BOOL;
   AntOffCh2_STN2 : BOOL;
   AntOffCh3_STN3 : BOOL;
   AntOffCh4_STN4 : BOOL;
   AUTO_STARTED : BOOL;
   AUTO_STARTED_STN1 : BOOL;
   AUTO_STARTED_STN2 : BOOL;
   AUTO_STARTED_STN3 : BOOL;
   AUTO_STARTED_STN4 : BOOL;
   BusyCh1 : BOOL;
   BusyCh1_STN1 : BOOL;
   BusyCh2 : BOOL;
   BusyCh2_STN2 : BOOL;
   BusyCh3_STN3 : BOOL;
   BusyCh4_STN4 : BOOL := 1;
   CH1_ONS : BOOL;
   Ch1Read : BOOL;
   Ch1Read_STN1 : BOOL;
   CH2_ON3 : BOOL;
   CH2_ON5_STN2 : BOOL := 1;
   CH2_ONS : BOOL;
   CH2_ONS3_STN2 : BOOL;
   CH2_ONS_STN2 : BOOL;
   Ch2Read : BOOL;
   Ch2Read_STN2 : BOOL;
   CH3_ON5_STN3 : BOOL := 1;
   CH3_ONS3_STN3 : BOOL;
   CH3_ONS_STN3 : BOOL;
   Ch3Read_STN3 : BOOL;
   CH4_ONS_STN4 : BOOL;
   Ch4Read_STN4 : BOOL;
   CRIMP_PASS_FROM_HP : DINT;
   DB_SAVED_OP20A : DINT; {produced}
   DB_SAVED_OP20B : DINT; {produced}
   DB_SAVED_OP20C : DINT; {produced}
   DB_SAVED_OP20D : DINT; {produced}
   DiagDataCh1 : DINT[4];
   DiagDataCh1_STN1 : DINT[4];
   DiagDataCh2 : DINT[4];
   DiagDataCh2_STN2 : DINT[4];
   DiagDataCh3_STN3 : DINT[4];
   DiagDataCh4_STN4 : DINT[4] := ([0] := 93388532);
   DiagLCh1 : INT;
   DiagLCh1_STN1 : INT;
   DiagLCh2 : INT;
   DiagLCh2_STN2 : INT;
   DiagLCh3_STN3 : INT;
   DiagLCh4_STN4 : INT := 1;
   DoneCh1 : BOOL;
   DoneCh1_STN1 : BOOL;
   DoneCh2 : BOOL;
   DoneCh2_STN2 : BOOL;
   DoneCh3_STN3 : BOOL;
   DoneCh4_STN4 : BOOL;
   DTE2_Status : DINT := 16384;
   DTE_ConnectionOK : BOOL := 1;
   DTE_ConnectionOK_2 : BOOL := 1;
   DTE_Status : DINT := 16384;
   dummit : BOOL;
   EMPTY_STRING : STRING;
   ErrorCh1 : BOOL;
   ErrorCh1_STN1 : BOOL;
   ErrorCh2 : BOOL;
   ErrorCh2_STN2 : BOOL;
   ErrorCh3_STN3 : BOOL;
   ErrorCh4_STN4 : BOOL;
   FLT_CLR_ONS_STN1 : DINT;
   FLT_CLR_ONS_STN2 : DINT;
   FLT_CLR_ONS_STN3 : DINT;
   FLT_CLR_ONS_STN4 : DINT;
   Generate_Rfid : BOOL;
   Generate_Rfid_Off_Del : TIMER := (PRE := 1000);
   HP_ACT_DROP_STN4 : REAL := 0.4958496;
   OP10_STATUS : INT;
   OP10_TAG_WRITE : BOOL;
   OP20A_DB_SAVED : BOOL;
   OP20A_DB_SAVED_DEL : TIMER := (PRE := 1000);
   OP20A_FAULTED : DINT := 2;
   OP20B_DB_SAVED : BOOL;
   OP20B_DB_SAVED_DEL : TIMER := (PRE := 1000);
   OP20B_FAULTED : DINT := 2;
   OP20C_DB_SAVED : BOOL;
   OP20C_DB_SAVED_DEL : TIMER := (PRE := 1000);
   OP20C_FAULTED : DINT := 2;
   OP20D_DB_SAVED : BOOL;
   OP20D_DB_SAVED_DEL : TIMER := (PRE := 1000);
   OP20D_FAULTED : DINT := 2;
   OP30_ACCEPT : BOOL;
   OP30_DB_SAVED : BOOL;
   OP30_DB_SAVED_DEL : TIMER := (PRE := 1000);
   OP30_REJECT : BOOL;
   OP30_STATUS : DINT;
   OVERALL_TRACE : BOOL;
   RcvBufCh1 : SINT[32];
   RcvBufCh1_STN1 : SINT[32];
   RcvBufCh2 : SINT[32];
   RcvBufCh2_STN2 : SINT[32];
   RcvBufCh3_STN3 : SINT[32];
   RcvBufCh4_STN4 : SINT[32];
   RcvdLCh1 : INT;
   RcvdLCh1_STN1 : INT;
   RcvdLCh2 : INT;
   RcvdLCh2_STN2 : INT;
   RcvdLCh3_STN3 : INT;
   RcvdLCh4_STN4 : INT;
   RdCh1 : BOOL;
   RdCh1_STN1 : BOOL;
   RdCh2 : BOOL;
   RdCh2_STN2 : BOOL;
   RdCh3_STN3 : BOOL;
   RdCh4_STN4 : BOOL;
   RdWrLengthCh1 : INT := 23;
   RdWrLengthCh1_STN1 : INT := 23;
   RdWrLengthCh2 : INT := 23;
   RdWrLengthCh2_STN2 : INT := 23;
   RdWrLengthCh3_STN3 : INT := 23;
   RdWrLengthCh4_STN4 : INT := 23;
   RdWrStartAddr_Ch2 : INT;
   RdWrStartAddr_STN1 : INT;
   RdWrStartAddr_STN2 : INT;
   RdWrStartAddr_STN3 : INT;
   RdWrStartAddr_STN4 : INT;
   READ_AGAIN_OP30 : BOOL;
   READ_AGAIN_STN1 : BOOL;
   READ_AGAIN_STN2 : BOOL;
   READ_AGAIN_STN3 : BOOL;
   READ_AGAIN_STN4 : BOOL;
   READ_DEL : TIMER := (PRE := 300);
   READ_DEL_OP30 : TIMER := (PRE := 300);
   READ_DEL_STN1 : TIMER := (PRE := 300);
   READ_DEL_STN2 : TIMER := (PRE := 300);
   READ_DEL_STN3 : TIMER := (PRE := 300);
   READ_DEL_STN4 : TIMER := (PRE := 300);
   REJECT_PB_OP30 : ALIAS FOR Local:1:I.Pt01.Data;
   RFID_GENERATED_1 : STRING := '2904712450Ch21122021002';
   RFID_HP : SINT[80];
   RFID_NI : STRING := '0029047352L0723Aj000018';
   RFID_OP30 : STRING := '0029047352L0723Aj000018';
   RWH_CH_1 : RWH_RW := (ixConnOK := 1, iiChannelNo := 3, ixUserMem := 1, iiRdWrLength := 23, owStatus := 16#0000_7000);
   RWH_CH_2 : RWH_RW := (ixConnOK := 1, iiChannelNo := 2, ixUserMem := 1, iiRdWrLength := 23, owStatus := 16#0000_7000);
   RWH_CH_4 : RWH_RW := (ixConnOK := 1, iiChannelNo := 4, oxBusy := 1, ixUserMem := 1, iiRdWrLength := 23, owStatus := 16#0000_7402, oiDiagLength := 1);
   RWH_CH_4_STN4 : RWH_RW := (ixConnOK := 1, iiChannelNo := 4, oxBusy := 1, ixUserMem := 1, iiRdWrLength := 23, owStatus := 16#0000_7403, oiDiagLength := 1);
   RWH_STN1 : RWH_RW := (ixConnOK := 1, iiChannelNo := 1, ixUserMem := 1, iiRdWrLength := 23, owStatus := 16#0000_7000);
   RWH_STN2 : RWH_RW := (ixConnOK := 1, iiChannelNo := 2, ixUserMem := 1, iiRdWrLength := 23, owStatus := 16#0000_7000);
   RWH_STN3 : RWH_RW := (ixConnOK := 1, iiChannelNo := 3, ixUserMem := 1, iiRdWrLength := 23, owStatus := 16#0000_7000);
   SendBufCh1 : SINT[32] := ([0] := 48, [1] := 48, [2] := 50, [3] := 57, [4] := 48, [5] := 52, [6] := 55, [7] := 51, [8] := 53, [9] := 50, [10] := 76, [11] := 48, [12] := 55, [13] := 50, [14] := 51, [15] := 65, [16] := 106, [17] := 48, [18] := 48, [19] := 48, [20] := 48, [21] := 49, [22] := 56);
   SendBufCh1_STN1 : SINT[32];
   SendBufCh2 : SINT[32];
   SendBufCh2_STN2 : SINT[32];
   SendBufCh3_STN3 : SINT[32];
   SendBufCh4_STN4 : SINT[32];
   so_Create_Instance : DINT := 1002;
   so_CreateParams : Createparams := (Type := 1, Addr.Family := 2, Addr.Port := 5002);
   so_write_Response : DINT := 10;
   so_WriteParams : WriteParams := (ToAddr.Family := 2, ToAddr.Port := 5020, Buf := 'TESTRIG50C');
   StatusCh1 : DINT := 16#0000_7000;
   StatusCh1_STN1 : DINT := 28672;
   StatusCh2 : DINT := 28672;
   StatusCh2_STN2 : DINT := 28672;
   StatusCh3_STN3 : DINT := 28672;
   StatusCh4_STN4 : DINT := 29699;
   STN1_RFID : STRING := '0029047352L0723Aj000018'; {produced}
   STN2_RFID : STRING; {produced}
   STN3_RFID : STRING; {produced}
   STN4_RFID : STRING; {produced}
   STS_OP_30 : DINT;
   TAG_CHANGE : DINT;
   Tag_Ind : INT;
   TAG_NOT_PRESENT_OP10 : BOOL;
   TAG_REMOVED_STN1 : TIMER := (PRE := 250, ACC := 250, EN := 1, DN := 1);
   TAG_REMOVED_STN2 : TIMER := (PRE := 500, ACC := 500, EN := 1, DN := 1);
   TAG_REMOVED_STN3 : TIMER := (PRE := 250, ACC := 250, EN := 1, DN := 1);
   TpCh1 : BOOL;
   TpCh1_STN1 : BOOL;
   TpCh2 : BOOL;
   TpCh2_STN2 : BOOL;
   TpCh3 : BOOL;
   TpCh3_STN3 : BOOL;
   TpCh4_STN4 : BOOL;
   TpCh5 : BOOL;
   TRACE_BYPASS_1 : BOOL;
   TRACE_ON : DINT[6] := ([4] := 1);
   TRACE_ON_STN1 : DINT := 1; {produced}
   TRACE_ON_STN2 : DINT := 1; {produced}
   TRACE_ON_STN3 : DINT := 1; {produced}
   TRACE_ON_STN4 : DINT := 1; {produced}
   TRACE_STATIONS : DINT := 15;
   TRACEABILITY_CY_START : DINT := 31;
   TS_STS_OP20A : DINT := 2; {produced}
   TS_STS_OP20B : DINT; {produced}
   TS_STS_OP20C : DINT; {produced}
   TS_STS_OP20D : DINT; {produced}
   TS_STS_OP30 : DINT;
   UrCh1 : BOOL := 1;
   UrCh1_STN1 : BOOL := 1;
   UrCh2 : BOOL := 1;
   UrCh2_STN2 : BOOL := 1;
   UrCh3_STN3 : BOOL := 1;
   UrCh4_STN4 : BOOL := 1;
   VEIFY_RFID : STRING := '0029047352L0717Dj000002'; {produced}
   WrCh1 : BOOL;
   WrCh1_STN1 : BOOL;
   WrCh2 : BOOL;
   WrCh2_STN2 : BOOL;
   WrCh3_STN3 : BOOL;
   WrCh4_STN4 : BOOL;
   WRITE : BOOL;
   WRITE_DEL : TIMER := (PRE := 1000);
END_VAR

PROGRAM MainProgram   (* main routine MainRoutine *)
VAR
   CH1_ON3 : BOOL;
   CH1_ON4 : BOOL;
   CH1_ON5 : BOOL := 1;
   CH1_ON5_STN1 : BOOL := 1;
   CH1_ONS3_STN1 : BOOL;
   CH1_ONS_STN1 : BOOL;
   CH2_ON5 : BOOL := 1;
   CH4_ON5_STN4 : BOOL := 1;
   CH4_ONS4_STN4 : BOOL;
   CRIMP_TAG_TIMEOUT : TIMER := (PRE := 2000);
   o_OFF_DE : TIMER := (PRE := 500);
   ONS1 : BOOL;
   ONS2 : BOOL;
   ONS3 : BOOL;
   ONS4 : BOOL;
   READ_AGAIN : BOOL;
   TAG_GEN_SEQ : DINT := 40;
   TS_OP20A_CLR_DEL : TIMER := (PRE := 500);
   WRITE_ON_DEL : TIMER := (PRE := 1000);
END_VAR

ROUTINE HP_TRACE   (* ladder *)
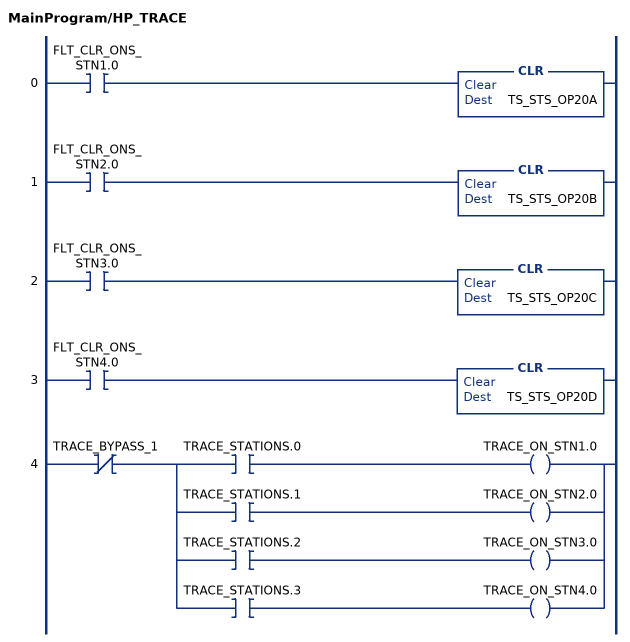
   0: XIC(FLT_CLR_ONS_STN1.0)CLR(TS_STS_OP20A);
   1: XIC(FLT_CLR_ONS_STN2.0)CLR(TS_STS_OP20B);
   2: XIC(FLT_CLR_ONS_STN3.0)CLR(TS_STS_OP20C);
   3: XIC(FLT_CLR_ONS_STN4.0)CLR(TS_STS_OP20D);
   4: XIO(TRACE_BYPASS_1)[XIC(TRACE_STATIONS.0) OTE(TRACE_ON_STN1.0) ,XIC(TRACE_STATIONS.1) OTE(TRACE_ON_STN2.0) ,XIC(TRACE_STATIONS.2) OTE(TRACE_ON_STN3.0) ,XIC(TRACE_STATIONS.3) OTE(TRACE_ON_STN4.0) ];
END_ROUTINE

ROUTINE MainRoutine   (* ladder *)
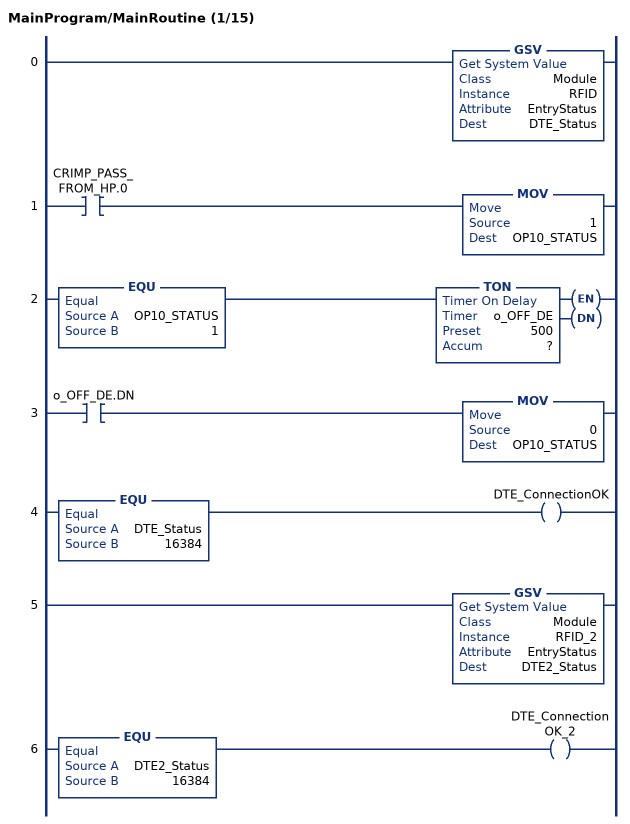
   0: GSV(Module,RFID,EntryStatus,DTE_Status);
   1: XIC(CRIMP_PASS_FROM_HP.0)MOV(1,OP10_STATUS);
   2: EQU(OP10_STATUS,1)TON(o_OFF_DE,?,?);
   3: XIC(o_OFF_DE.DN)MOV(0,OP10_STATUS);
   4: EQU(DTE_Status,16384)OTE(DTE_ConnectionOK);
   5: GSV(Module,RFID_2,EntryStatus,DTE2_Status);
   6: EQU(DTE2_Status,16384)OTE(DTE_ConnectionOK_2);
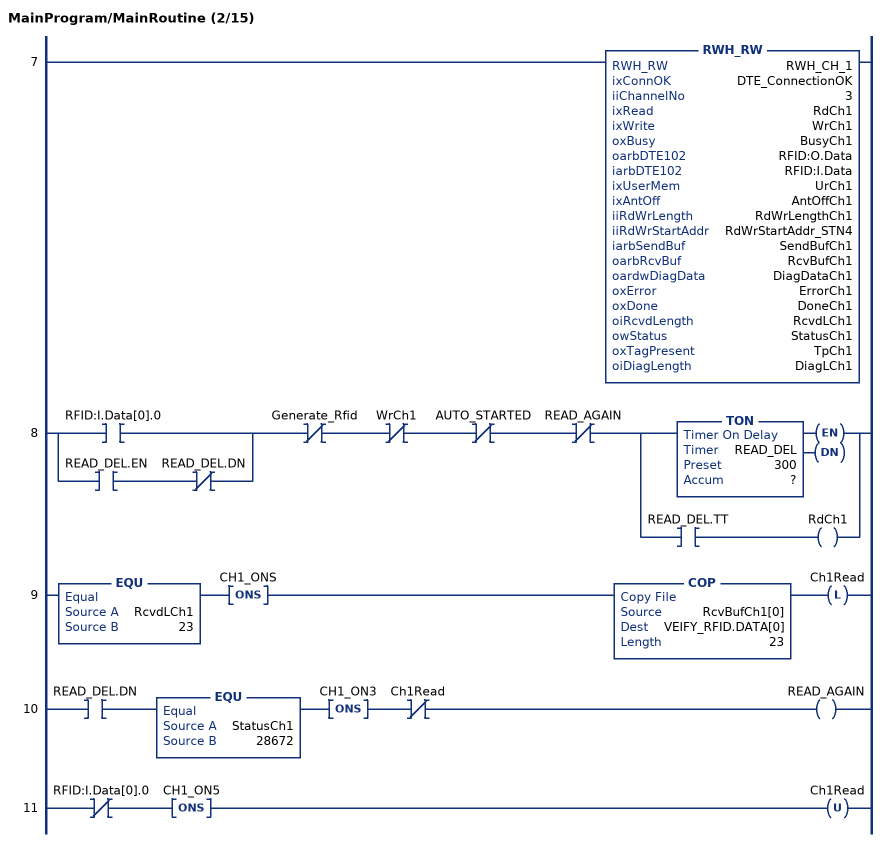
   7: RWH_RW(RWH_CH_1,DTE_ConnectionOK,3,RdCh1,WrCh1,BusyCh1,RFID:O.Data,RFID:I.Data,UrCh1,AntOffCh1,RdWrLengthCh1,RdWrStartAddr_STN4,SendBufCh1,RcvBufCh1,DiagDataCh1,ErrorCh1,DoneCh1,RcvdLCh1,StatusCh1,TpCh1,DiagLCh1);
   8: [XIC(RFID:I.Data[0].0) ,XIC(READ_DEL.EN) XIO(READ_DEL.DN) ]XIO(Generate_Rfid)XIO(WrCh1)XIO(AUTO_STARTED)XIO(READ_AGAIN)[TON(READ_DEL,?,?) ,XIC(READ_DEL.TT) OTE(RdCh1) ];
   9: EQU(RcvdLCh1,23)ONS(CH1_ONS)COP(RcvBufCh1[0],VEIFY_RFID.DATA[0],23)OTL(Ch1Read);
   10: XIC(READ_DEL.DN)EQU(StatusCh1,28672)ONS(CH1_ON3)XIO(Ch1Read)OTE(READ_AGAIN);
   11: XIO(RFID:I.Data[0].0)ONS(CH1_ON5)OTU(Ch1Read);
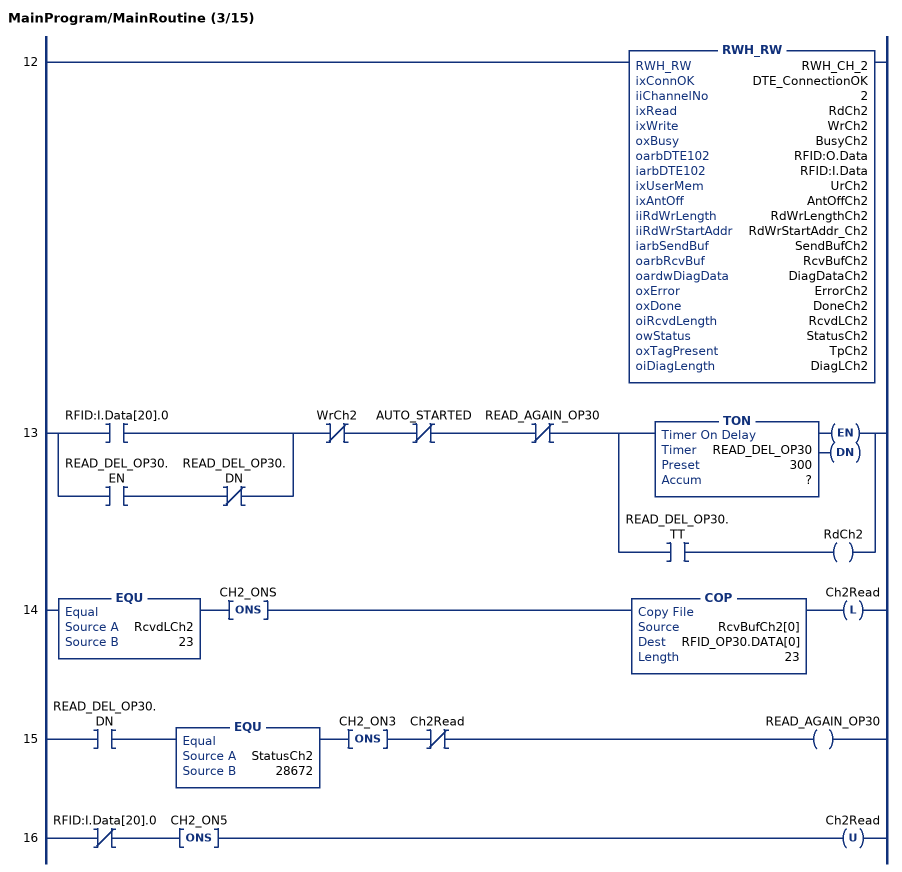
   12: RWH_RW(RWH_CH_2,DTE_ConnectionOK,2,RdCh2,WrCh2,BusyCh2,RFID:O.Data,RFID:I.Data,UrCh2,AntOffCh2,RdWrLengthCh2,RdWrStartAddr_Ch2,SendBufCh2,RcvBufCh2,DiagDataCh2,ErrorCh2,DoneCh2,RcvdLCh2,StatusCh2,TpCh2,DiagLCh2);
   13: [XIC(RFID:I.Data[20].0) ,XIC(READ_DEL_OP30.EN) XIO(READ_DEL_OP30.DN) ]XIO(WrCh2)XIO(AUTO_STARTED)XIO(READ_AGAIN_OP30)[TON(READ_DEL_OP30,?,?) ,XIC(READ_DEL_OP30.TT) OTE(RdCh2) ];
   14: EQU(RcvdLCh2,23)ONS(CH2_ONS)COP(RcvBufCh2[0],RFID_OP30.DATA[0],23)OTL(Ch2Read);
   15: XIC(READ_DEL_OP30.DN)EQU(StatusCh2,28672)ONS(CH2_ON3)XIO(Ch2Read)OTE(READ_AGAIN_OP30);
   16: XIO(RFID:I.Data[20].0)ONS(CH2_ON5)OTU(Ch2Read);
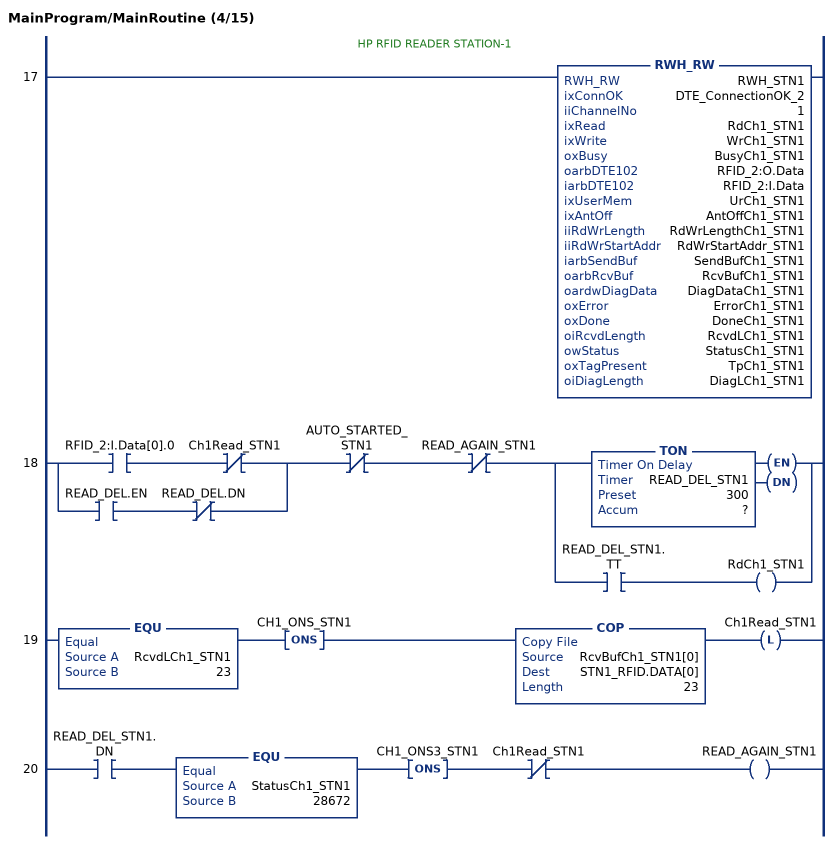
   // HP RFID READER STATION-1
   17: RWH_RW(RWH_STN1,DTE_ConnectionOK_2,1,RdCh1_STN1,WrCh1_STN1,BusyCh1_STN1,RFID_2:O.Data,RFID_2:I.Data,UrCh1_STN1,AntOffCh1_STN1,RdWrLengthCh1_STN1,RdWrStartAddr_STN1,SendBufCh1_STN1,RcvBufCh1_STN1,DiagDataCh1_STN1,ErrorCh1_STN1,DoneCh1_STN1,RcvdLCh1_STN1,StatusCh1_STN1,TpCh1_STN1,DiagLCh1_STN1);
   18: [XIC(RFID_2:I.Data[0].0) XIO(Ch1Read_STN1) ,XIC(READ_DEL.EN) XIO(READ_DEL.DN) ]XIO(AUTO_STARTED_STN1)XIO(READ_AGAIN_STN1)[TON(READ_DEL_STN1,?,?) ,XIC(READ_DEL_STN1.TT) OTE(RdCh1_STN1) ];
   19: EQU(RcvdLCh1_STN1,23)ONS(CH1_ONS_STN1)COP(RcvBufCh1_STN1[0],STN1_RFID.DATA[0],23)OTL(Ch1Read_STN1);
   20: XIC(READ_DEL_STN1.DN)EQU(StatusCh1_STN1,28672)ONS(CH1_ONS3_STN1)XIO(Ch1Read_STN1)OTE(READ_AGAIN_STN1);
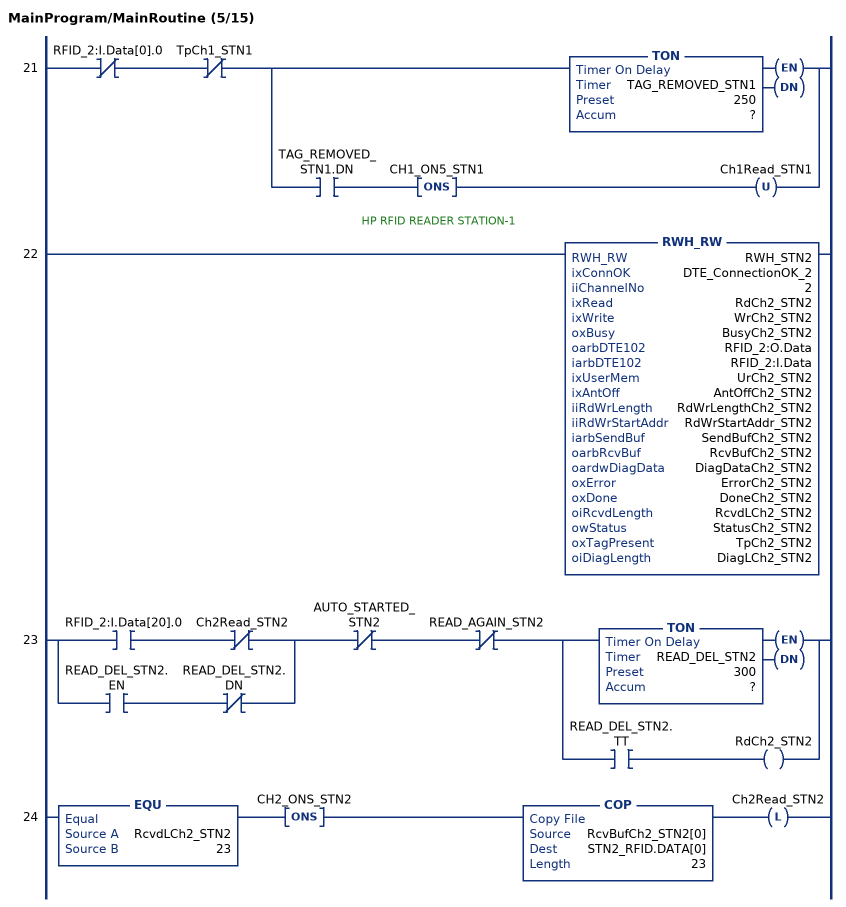
   21: XIO(RFID_2:I.Data[0].0)XIO(TpCh1_STN1)[TON(TAG_REMOVED_STN1,?,?) ,XIC(TAG_REMOVED_STN1.DN) ONS(CH1_ON5_STN1) OTU(Ch1Read_STN1) ];
   // HP RFID READER STATION-1
   22: RWH_RW(RWH_STN2,DTE_ConnectionOK_2,2,RdCh2_STN2,WrCh2_STN2,BusyCh2_STN2,RFID_2:O.Data,RFID_2:I.Data,UrCh2_STN2,AntOffCh2_STN2,RdWrLengthCh2_STN2,RdWrStartAddr_STN2,SendBufCh2_STN2,RcvBufCh2_STN2,DiagDataCh2_STN2,ErrorCh2_STN2,DoneCh2_STN2,RcvdLCh2_STN2,StatusCh2_STN2,TpCh2_STN2,DiagLCh2_STN2);
   23: [XIC(RFID_2:I.Data[20].0) XIO(Ch2Read_STN2) ,XIC(READ_DEL_STN2.EN) XIO(READ_DEL_STN2.DN) ]XIO(AUTO_STARTED_STN2)XIO(READ_AGAIN_STN2)[TON(READ_DEL_STN2,?,?) ,XIC(READ_DEL_STN2.TT) OTE(RdCh2_STN2) ];
   24: EQU(RcvdLCh2_STN2,23)ONS(CH2_ONS_STN2)COP(RcvBufCh2_STN2[0],STN2_RFID.DATA[0],23)OTL(Ch2Read_STN2);
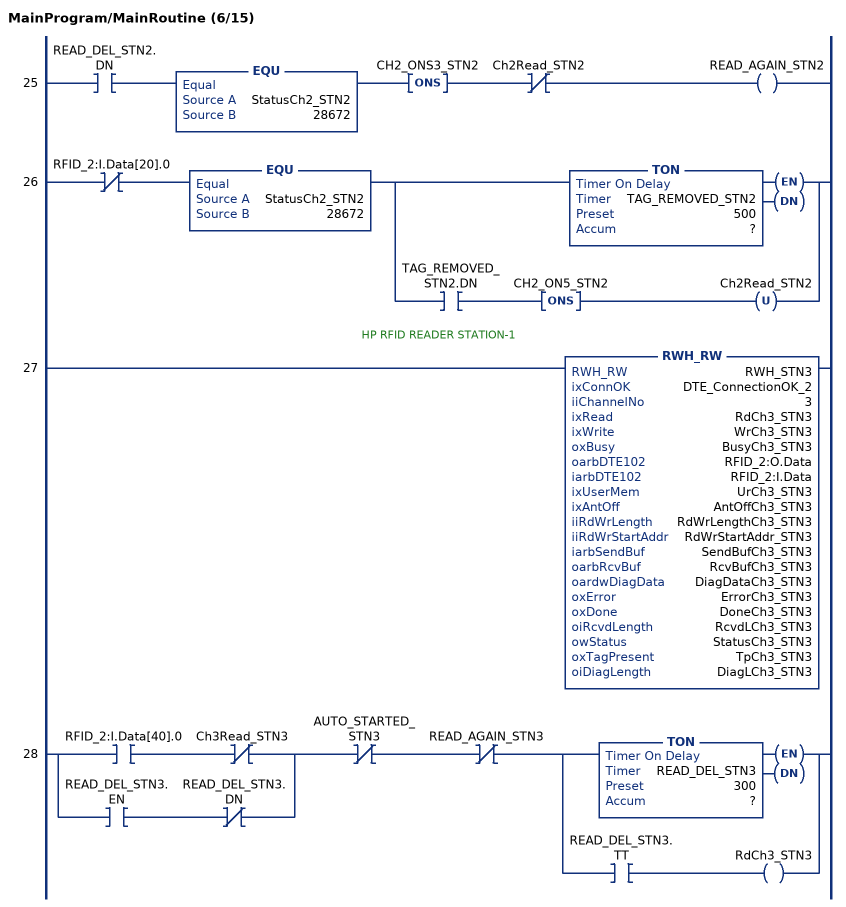
   25: XIC(READ_DEL_STN2.DN)EQU(StatusCh2_STN2,28672)ONS(CH2_ONS3_STN2)XIO(Ch2Read_STN2)OTE(READ_AGAIN_STN2);
   26: XIO(RFID_2:I.Data[20].0)EQU(StatusCh2_STN2,28672)[TON(TAG_REMOVED_STN2,?,?) ,XIC(TAG_REMOVED_STN2.DN) ONS(CH2_ON5_STN2) OTU(Ch2Read_STN2) ];
   // HP RFID READER STATION-1
   27: RWH_RW(RWH_STN3,DTE_ConnectionOK_2,3,RdCh3_STN3,WrCh3_STN3,BusyCh3_STN3,RFID_2:O.Data,RFID_2:I.Data,UrCh3_STN3,AntOffCh3_STN3,RdWrLengthCh3_STN3,RdWrStartAddr_STN3,SendBufCh3_STN3,RcvBufCh3_STN3,DiagDataCh3_STN3,ErrorCh3_STN3,DoneCh3_STN3,RcvdLCh3_STN3,StatusCh3_STN3,TpCh3_STN3,DiagLCh3_STN3);
   28: [XIC(RFID_2:I.Data[40].0) XIO(Ch3Read_STN3) ,XIC(READ_DEL_STN3.EN) XIO(READ_DEL_STN3.DN) ]XIO(AUTO_STARTED_STN3)XIO(READ_AGAIN_STN3)[TON(READ_DEL_STN3,?,?) ,XIC(READ_DEL_STN3.TT) OTE(RdCh3_STN3) ];
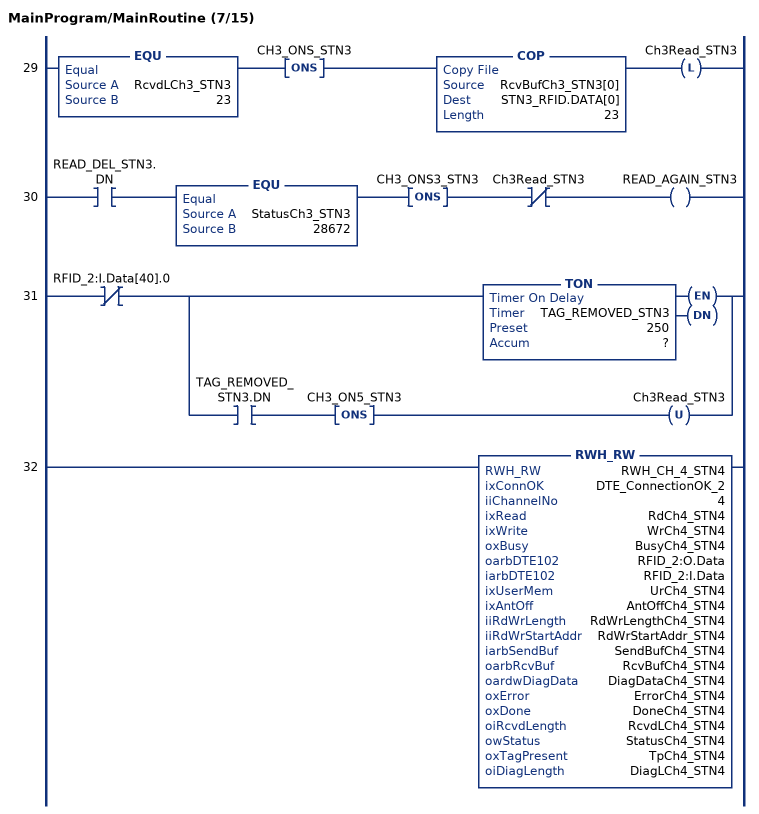
   29: EQU(RcvdLCh3_STN3,23)ONS(CH3_ONS_STN3)COP(RcvBufCh3_STN3[0],STN3_RFID.DATA[0],23)OTL(Ch3Read_STN3);
   30: XIC(READ_DEL_STN3.DN)EQU(StatusCh3_STN3,28672)ONS(CH3_ONS3_STN3)XIO(Ch3Read_STN3)OTE(READ_AGAIN_STN3);
   31: XIO(RFID_2:I.Data[40].0)[TON(TAG_REMOVED_STN3,?,?) ,XIC(TAG_REMOVED_STN3.DN) ONS(CH3_ON5_STN3) OTU(Ch3Read_STN3) ];
   32: RWH_RW(RWH_CH_4_STN4,DTE_ConnectionOK_2,4,RdCh4_STN4,WrCh4_STN4,BusyCh4_STN4,RFID_2:O.Data,RFID_2:I.Data,UrCh4_STN4,AntOffCh4_STN4,RdWrLengthCh4_STN4,RdWrStartAddr_STN4,SendBufCh4_STN4,RcvBufCh4_STN4,DiagDataCh4_STN4,ErrorCh4_STN4,DoneCh4_STN4,RcvdLCh4_STN4,StatusCh4_STN4,TpCh4_STN4,DiagLCh4_STN4);
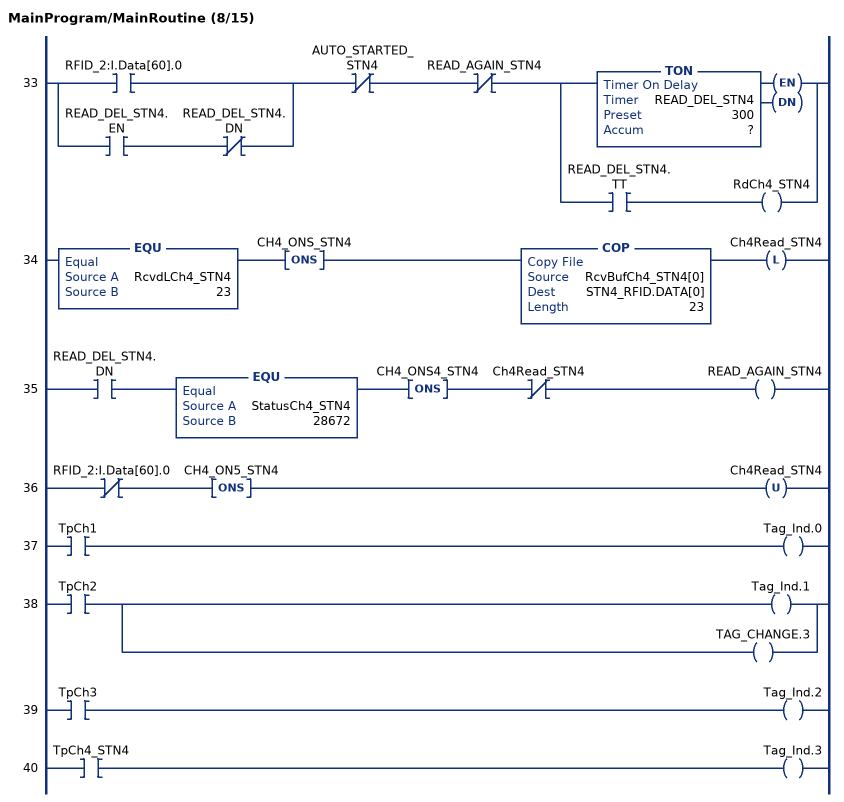
   33: [XIC(RFID_2:I.Data[60].0) ,XIC(READ_DEL_STN4.EN) XIO(READ_DEL_STN4.DN) ]XIO(AUTO_STARTED_STN4)XIO(READ_AGAIN_STN4)[TON(READ_DEL_STN4,?,?) ,XIC(READ_DEL_STN4.TT) OTE(RdCh4_STN4) ];
   34: EQU(RcvdLCh4_STN4,23)ONS(CH4_ONS_STN4)COP(RcvBufCh4_STN4[0],STN4_RFID.DATA[0],23)OTL(Ch4Read_STN4);
   35: XIC(READ_DEL_STN4.DN)EQU(StatusCh4_STN4,28672)ONS(CH4_ONS4_STN4)XIO(Ch4Read_STN4)OTE(READ_AGAIN_STN4);
   36: XIO(RFID_2:I.Data[60].0)ONS(CH4_ON5_STN4)OTU(Ch4Read_STN4);
   37: XIC(TpCh1)OTE(Tag_Ind.0);
   38: XIC(TpCh2)[OTE(Tag_Ind.1) ,OTE(TAG_CHANGE.3) ];
   39: XIC(TpCh3)OTE(Tag_Ind.2);
   40: XIC(TpCh4_STN4)OTE(Tag_Ind.3);
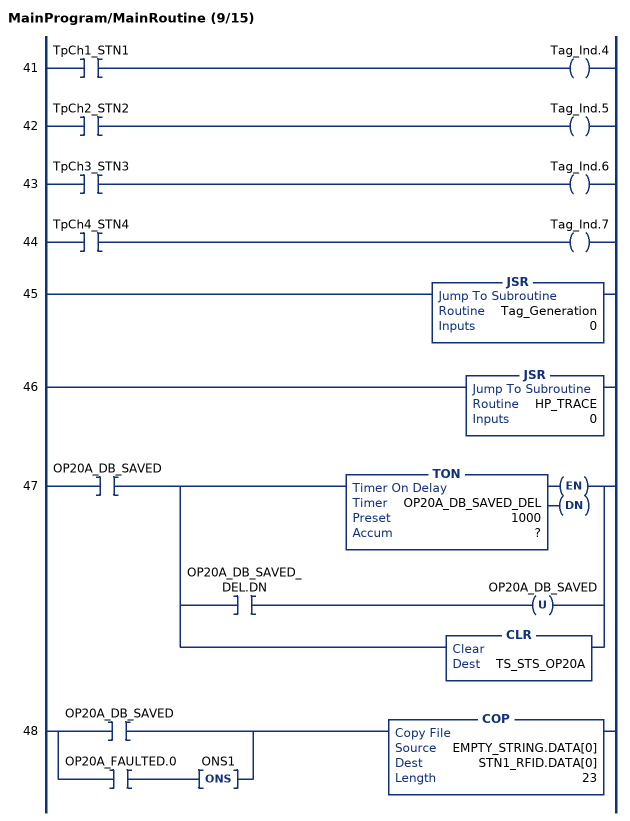
   41: XIC(TpCh1_STN1)OTE(Tag_Ind.4);
   42: XIC(TpCh2_STN2)OTE(Tag_Ind.5);
   43: XIC(TpCh3_STN3)OTE(Tag_Ind.6);
   44: XIC(TpCh4_STN4)OTE(Tag_Ind.7);
   45: JSR(Tag_Generation,0);
   46: JSR(HP_TRACE,0);
   47: XIC(OP20A_DB_SAVED)[TON(OP20A_DB_SAVED_DEL,?,?) ,XIC(OP20A_DB_SAVED_DEL.DN) OTU(OP20A_DB_SAVED) ,CLR(TS_STS_OP20A) ];
   48: [XIC(OP20A_DB_SAVED) ,XIC(OP20A_FAULTED.0) ONS(ONS1) ]COP(EMPTY_STRING.DATA[0],STN1_RFID.DATA[0],23);
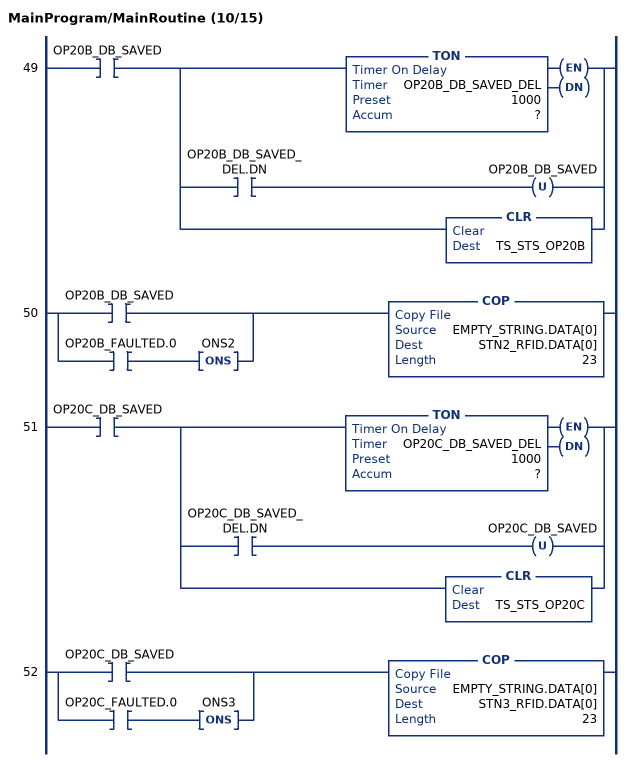
   49: XIC(OP20B_DB_SAVED)[TON(OP20B_DB_SAVED_DEL,?,?) ,XIC(OP20B_DB_SAVED_DEL.DN) OTU(OP20B_DB_SAVED) ,CLR(TS_STS_OP20B) ];
   50: [XIC(OP20B_DB_SAVED) ,XIC(OP20B_FAULTED.0) ONS(ONS2) ]COP(EMPTY_STRING.DATA[0],STN2_RFID.DATA[0],23);
   51: XIC(OP20C_DB_SAVED)[TON(OP20C_DB_SAVED_DEL,?,?) ,XIC(OP20C_DB_SAVED_DEL.DN) OTU(OP20C_DB_SAVED) ,CLR(TS_STS_OP20C) ];
   52: [XIC(OP20C_DB_SAVED) ,XIC(OP20C_FAULTED.0) ONS(ONS3) ]COP(EMPTY_STRING.DATA[0],STN3_RFID.DATA[0],23);
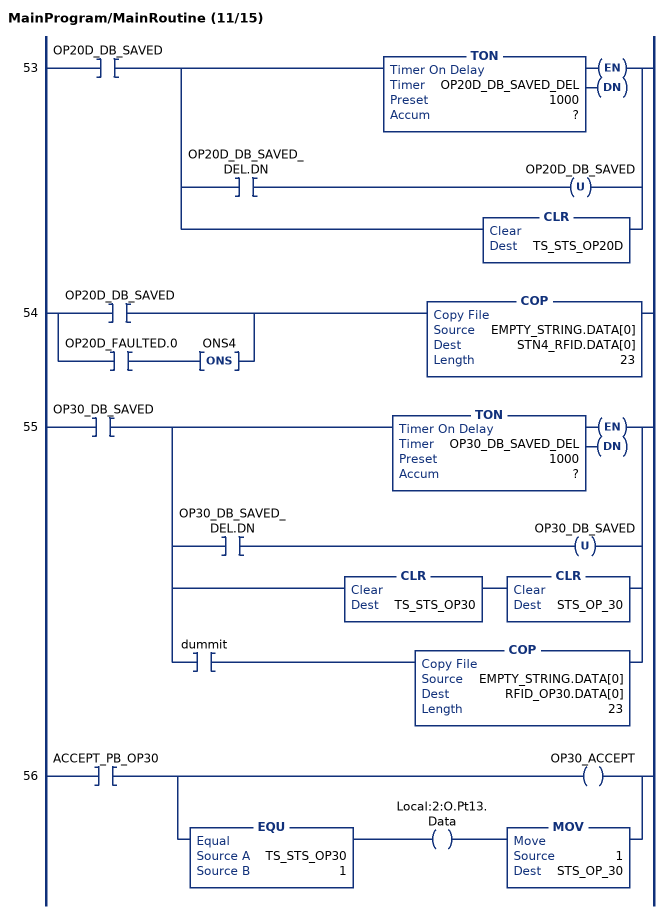
   53: XIC(OP20D_DB_SAVED)[TON(OP20D_DB_SAVED_DEL,?,?) ,XIC(OP20D_DB_SAVED_DEL.DN) OTU(OP20D_DB_SAVED) ,CLR(TS_STS_OP20D) ];
   54: [XIC(OP20D_DB_SAVED) ,XIC(OP20D_FAULTED.0) ONS(ONS4) ]COP(EMPTY_STRING.DATA[0],STN4_RFID.DATA[0],23);
   55: XIC(OP30_DB_SAVED)[TON(OP30_DB_SAVED_DEL,?,?) ,XIC(OP30_DB_SAVED_DEL.DN) OTU(OP30_DB_SAVED) ,CLR(TS_STS_OP30) CLR(STS_OP_30) ,XIC(dummit) COP(EMPTY_STRING.DATA[0],RFID_OP30.DATA[0],23) ];
   56: XIC(ACCEPT_PB_OP30)[OTE(OP30_ACCEPT) ,EQU(TS_STS_OP30,1) OTE(Local:2:O.Pt13.Data) MOV(1,STS_OP_30) ];
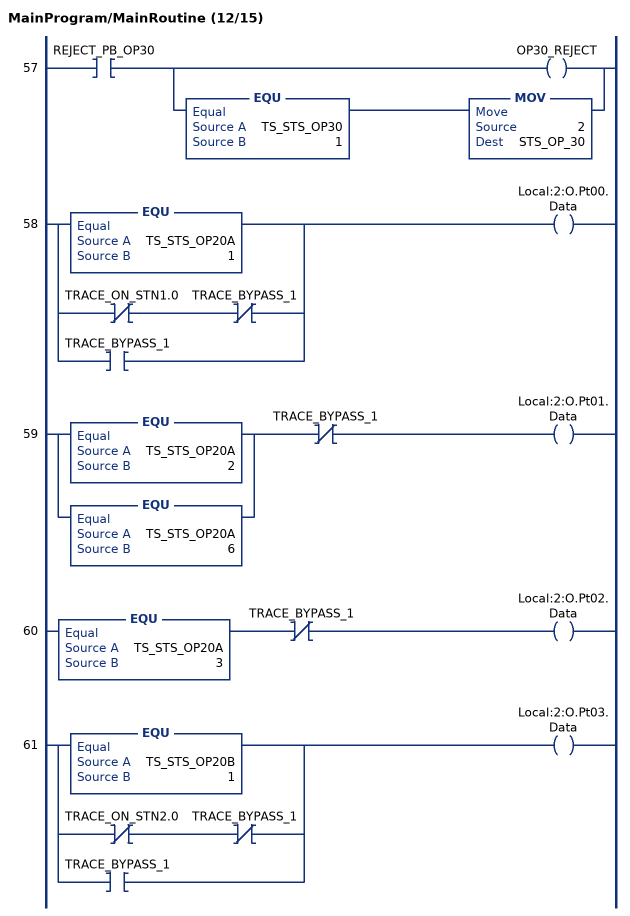
   57: XIC(REJECT_PB_OP30)[OTE(OP30_REJECT) ,EQU(TS_STS_OP30,1) MOV(2,STS_OP_30) ];
   58: [EQU(TS_STS_OP20A,1) ,XIO(TRACE_ON_STN1.0) XIO(TRACE_BYPASS_1) ,XIC(TRACE_BYPASS_1) ]OTE(Local:2:O.Pt00.Data);
   59: [EQU(TS_STS_OP20A,2) ,EQU(TS_STS_OP20A,6) ]XIO(TRACE_BYPASS_1)OTE(Local:2:O.Pt01.Data);
   60: EQU(TS_STS_OP20A,3)XIO(TRACE_BYPASS_1)OTE(Local:2:O.Pt02.Data);
   61: [EQU(TS_STS_OP20B,1) ,XIO(TRACE_ON_STN2.0) XIO(TRACE_BYPASS_1) ,XIC(TRACE_BYPASS_1) ]OTE(Local:2:O.Pt03.Data);
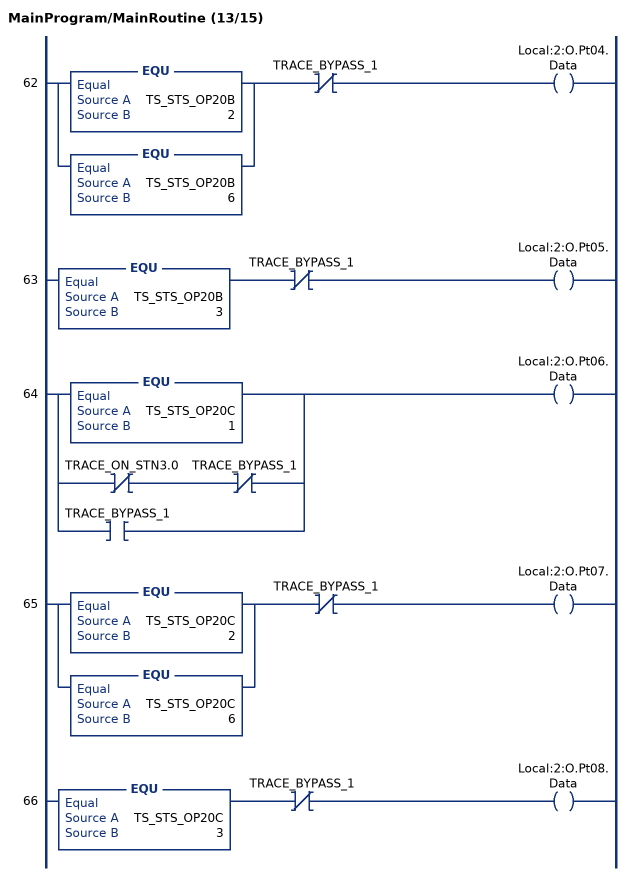
   62: [EQU(TS_STS_OP20B,2) ,EQU(TS_STS_OP20B,6) ]XIO(TRACE_BYPASS_1)OTE(Local:2:O.Pt04.Data);
   63: EQU(TS_STS_OP20B,3)XIO(TRACE_BYPASS_1)OTE(Local:2:O.Pt05.Data);
   64: [EQU(TS_STS_OP20C,1) ,XIO(TRACE_ON_STN3.0) XIO(TRACE_BYPASS_1) ,XIC(TRACE_BYPASS_1) ]OTE(Local:2:O.Pt06.Data);
   65: [EQU(TS_STS_OP20C,2) ,EQU(TS_STS_OP20C,6) ]XIO(TRACE_BYPASS_1)OTE(Local:2:O.Pt07.Data);
   66: EQU(TS_STS_OP20C,3)XIO(TRACE_BYPASS_1)OTE(Local:2:O.Pt08.Data);
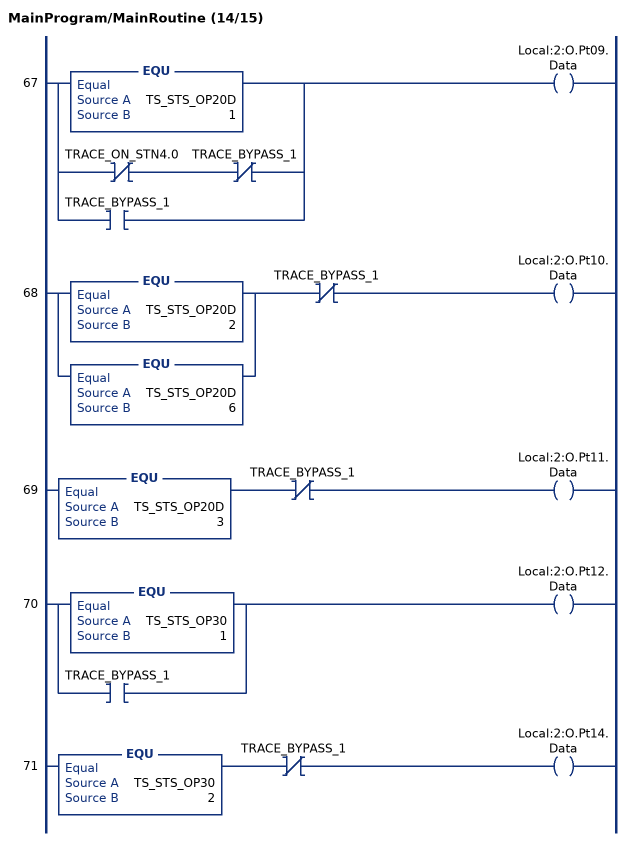
   67: [EQU(TS_STS_OP20D,1) ,XIO(TRACE_ON_STN4.0) XIO(TRACE_BYPASS_1) ,XIC(TRACE_BYPASS_1) ]OTE(Local:2:O.Pt09.Data);
   68: [EQU(TS_STS_OP20D,2) ,EQU(TS_STS_OP20D,6) ]XIO(TRACE_BYPASS_1)OTE(Local:2:O.Pt10.Data);
   69: EQU(TS_STS_OP20D,3)XIO(TRACE_BYPASS_1)OTE(Local:2:O.Pt11.Data);
   70: [EQU(TS_STS_OP30,1) ,XIC(TRACE_BYPASS_1) ]OTE(Local:2:O.Pt12.Data);
   71: EQU(TS_STS_OP30,2)XIO(TRACE_BYPASS_1)OTE(Local:2:O.Pt14.Data);
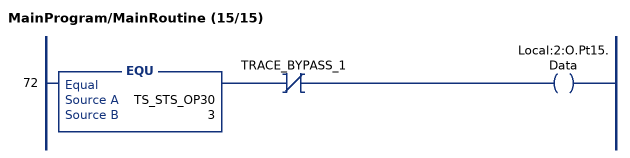
   72: EQU(TS_STS_OP30,3)XIO(TRACE_BYPASS_1)OTE(Local:2:O.Pt15.Data);
END_ROUTINE

ROUTINE Tag_Generation   (* ladder *)
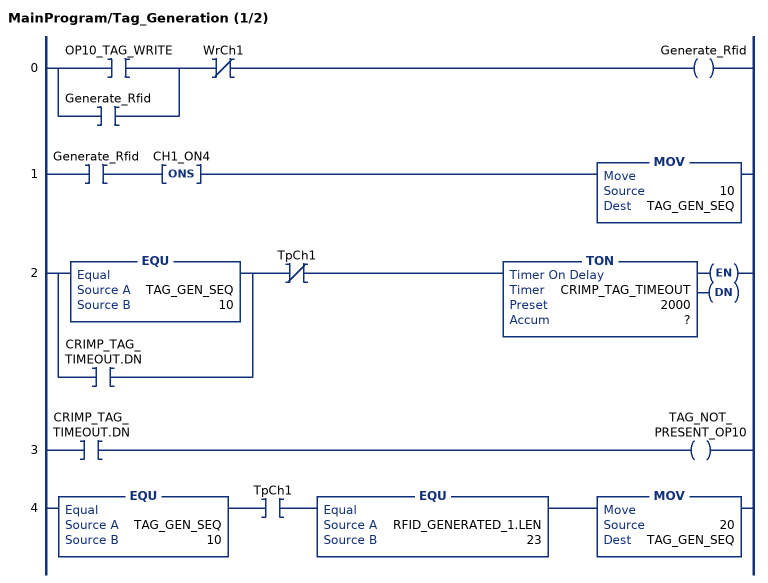
   0: [XIC(OP10_TAG_WRITE) ,XIC(Generate_Rfid) ]XIO(WrCh1)OTE(Generate_Rfid);
   1: XIC(Generate_Rfid)ONS(CH1_ON4)MOV(10,TAG_GEN_SEQ);
   2: [EQU(TAG_GEN_SEQ,10) ,XIC(CRIMP_TAG_TIMEOUT.DN) ]XIO(TpCh1)TON(CRIMP_TAG_TIMEOUT,?,?);
   3: XIC(CRIMP_TAG_TIMEOUT.DN)OTE(TAG_NOT_PRESENT_OP10);
   4: EQU(TAG_GEN_SEQ,10)XIC(TpCh1)EQU(RFID_GENERATED_1.LEN,23)MOV(20,TAG_GEN_SEQ);
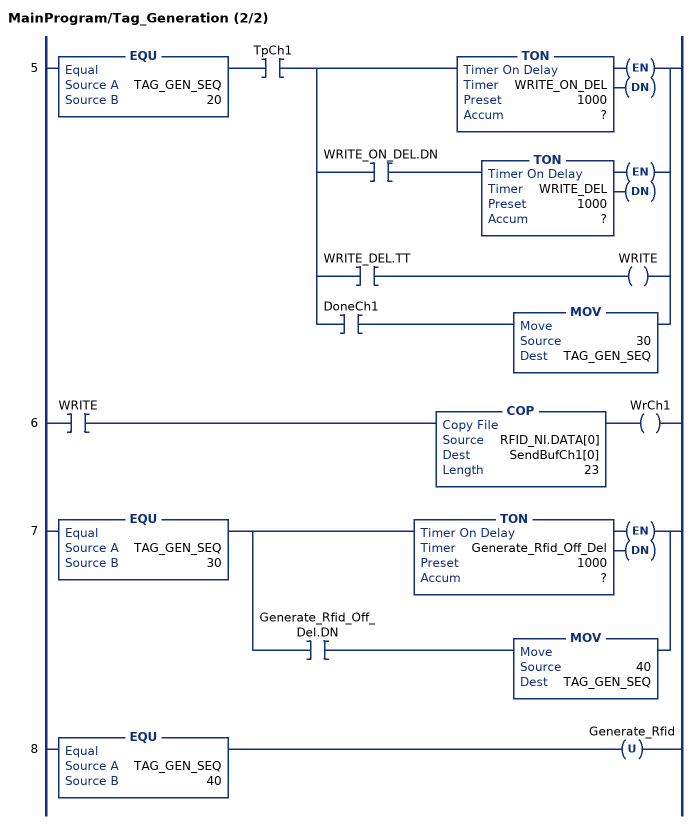
   5: EQU(TAG_GEN_SEQ,20)XIC(TpCh1)[TON(WRITE_ON_DEL,?,?) ,XIC(WRITE_ON_DEL.DN) TON(WRITE_DEL,?,?) ,XIC(WRITE_DEL.TT) OTE(WRITE) ,XIC(DoneCh1) MOV(30,TAG_GEN_SEQ) ];
   6: XIC(WRITE)COP(RFID_NI.DATA[0],SendBufCh1[0],23)OTE(WrCh1);
   7: EQU(TAG_GEN_SEQ,30)[TON(Generate_Rfid_Off_Del,?,?) ,XIC(Generate_Rfid_Off_Del.DN) MOV(40,TAG_GEN_SEQ) ];
   8: EQU(TAG_GEN_SEQ,40)OTU(Generate_Rfid);
END_ROUTINE
END_PROGRAM
